C07313=1200.137,5.931,-43.793,-179.713,5.631,148.907
C07314=1200.132,6.181,-43.807,-179.710,5.632,148.906
C07315=1200.127,6.431,-43.821,-179.708,5.632,148.906
C07316=1200.122,6.680,-43.836,-179.705,5.633,148.905
C07317=1200.117,6.929,-43.850,-179.703,5.633,148.904
C07318=1200.112,7.178,-43.865,-179.701,5.633,148.904
C07319=1200.107,7.428,-43.879,-179.698,5.634,148.903
C07320=1200.102,7.678,-43.893,-179.695,5.634,148.902
C07321=1200.097,7.928,-43.907,-179.693,5.635,148.902
C07322=1200.091,8.177,-43.921,-179.691,5.635,148.901
C07323=1200.086,8.426,-43.936,-179.688,5.636,148.900
C07324=1200.081,8.676,-43.950,-179.685,5.636,148.900
C07325=1200.076,8.926,-43.964,-179.683,5.637,148.899
C07326=1200.071,9.175,-43.978,-179.680,5.637,148.898
C07327=1200.066,9.425,-43.993,-179.678,5.638,148.898
C07328=1200.061,9.674,-44.007,-179.675,5.639,148.897
C07329=1200.056,9.923,-44.022,-179.673,5.639,148.897
C07330=1200.051,10.173,-44.036,-179.670,5.639,148.896
C07331=1200.046,10.423,-44.050,-179.668,5.640,148.895
C07332=1200.041,10.673,-44.065,-179.666,5.640,148.895
C07333=1200.036,10.922,-44.079,-179.663,5.641,148.894
C07334=1200.031,11.172,-44.094,-179.660,5.641,148.893
C07335=1200.026,11.421,-44.108,-179.658,5.642,148.893
C07336=1200.021,11.670,-44.123,-179.655,5.642,148.892
C07337=1200.016,11.920,-44.137,-179.652,5.643,148.891
C07338=1200.011,12.170,-44.151,-179.650,5.644,148.891
C07339=1200.006,12.419,-44.166,-179.648,5.644,148.890
C07340=1200.001,12.668,-44.180,-179.645,5.645,148.890
C07341=1199.995,12.918,-44.195,-179.642,5.645,148.889
C07342=1199.990,13.168,-44.210,-179.640,5.646,148.888
C07343=1199.986,13.417,-44.225,-179.637,5.647,148.888
C07344=1199.980,13.666,-44.238,-179.635,5.646,148.887
C07345=1199.975,13.916,-44.253,-179.633,5.647,148.886
C07346=1199.970,14.166,-44.267,-179.630,5.647,148.886
C07347=1199.966,14.415,-44.282,-179.627,5.648,148.885
C07348=1199.960,14.665,-44.297,-179.625,5.649,148.885
C07349=1199.955,14.915,-44.311,-179.623,5.649,148.884
C07350=1199.950,15.164,-44.326,-179.620,5.650,148.883
C07351=1199.945,15.413,-44.340,-179.617,5.650,148.882
C07352=1199.940,15.663,-44.355,-179.615,5.651,148.882
C07353=1199.935,15.912,-44.370,-179.613,5.652,148.881
C07354=1199.930,16.162,-44.385,-179.610,5.652,148.881
C07355=1199.925,16.412,-44.399,-179.607,5.653,148.880
C07356=1199.920,16.661,-44.414,-179.605,5.653,148.879
C07357=1199.916,16.911,-44.428,-179.602,5.654,148.879
C07358=1199.910,17.161,-44.443,-179.600,5.655,148.878
C07359=1199.905,17.410,-44.458,-179.597,5.655,148.877
C07360=1199.900,17.659,-44.472,-179.594,5.656,148.877
C07361=1199.895,17.908,-44.487,-179.592,5.656,148.876
C07362=1199.889,18.158,-44.502,-179.589,5.657,148.875
C07363=1199.884,18.408,-44.516,-179.587,5.657,148.875
C07364=1199.880,18.657,-44.531,-179.584,5.658,148.874
C07365=1199.875,18.906,-44.545,-179.582,5.658,148.874
C07366=1199.869,19.156,-44.561,-179.580,5.658,148.873
C07367=1199.864,19.406,-44.575,-179.577,5.659,148.872
C07368=1199.860,19.655,-44.590,-179.575,5.660,148.872
C07369=1199.854,19.905,-44.605,-179.572,5.660,148.871
C07370=1199.849,20.154,-44.620,-179.570,5.661,148.870
C07371=1199.844,20.403,-44.634,-179.567,5.661,148.870
C07372=1199.839,20.653,-44.650,-179.564,5.662,148.869
C07373=1199.834,20.903,-44.664,-179.562,5.662,148.869
C07374=1199.829,21.152,-44.679,-179.559,5.663,148.868
C07375=1199.824,21.402,-44.694,-179.557,5.663,148.867
C07376=1199.819,21.651,-44.709,-179.554,5.664,148.867
C07377=1199.814,21.900,-44.723,-179.552,5.665,148.866
C07378=1199.809,22.151,-44.739,-179.549,5.665,148.865
C07379=1199.804,22.400,-44.754,-179.547,5.666,148.865
C07380=1199.800,22.649,-44.768,-179.544,5.666,148.864
C07381=1199.794,22.899,-44.783,-179.541,5.667,148.863
C07382=1199.789,23.149,-44.798,-179.539,5.668,148.863
C07383=1199.785,23.398,-44.813,-179.537,5.668,148.862
C07384=1199.779,23.648,-44.828,-179.534,5.669,148.862
C07385=1199.774,23.897,-44.843,-179.531,5.669,148.861
C07386=1199.769,24.147,-44.858,-179.529,5.670,148.860
C07387=1199.764,24.396,-44.873,-179.527,5.671,148.860
C07388=1199.759,24.645,-44.888,-179.524,5.671,148.859
C07389=1199.754,24.895,-44.903,-179.521,5.672,148.858
C07390=1199.749,25.144,-44.918,-179.519,5.672,148.858
C07391=1199.744,25.393,-44.934,-179.516,5.673,148.857
C07392=1199.739,25.643,-44.948,-179.514,5.674,148.857
C07393=1199.735,25.893,-44.963,-179.511,5.674,148.856
C07394=1199.729,26.142,-44.979,-179.508,5.675,148.855
C07395=1199.724,26.392,-44.993,-179.506,5.675,148.855
C07396=1199.719,26.641,-45.009,-179.504,5.676,148.854
C07397=1199.714,26.891,-45.024,-179.501,5.677,148.853
C07398=1199.709,27.141,-45.038,-179.498,5.677,148.853
C07399=1199.704,27.390,-45.053,-179.496,5.678,148.852
C07400=1199.699,27.639,-45.069,-179.494,5.678,148.852
C07401=1199.694,27.888,-45.084,-179.491,5.679,148.851
C07402=1199.689,28.139,-45.099,-179.488,5.680,148.850
C07403=1199.684,28.388,-45.114,-179.486,5.680,148.850
C07404=1199.679,28.656,-45.131,-179.483,5.681,148.849
C07405=1199.674,28.925,-45.147,-179.480,5.681,148.848
C07406=1199.668,29.194,-45.163,-179.478,5.682,148.848
C07407=1199.663,29.462,-45.180,-179.474,5.683,148.847
C07408=1199.657,29.712,-45.195,-179.472,5.684,148.846
C07409=1199.653,29.962,-45.210,-179.470,5.684,148.846
C07410=1199.647,30.211,-45.225,-179.467,5.685,148.845
C07411=1199.642,30.460,-45.241,-179.464,5.685,148.844
C07412=1199.638,30.710,-45.256,-179.462,5.686,148.844
C07413=1199.632,30.960,-45.272,-179.460,5.687,148.843
C07414=1199.628,31.209,-45.287,-179.457,5.687,148.843
C07415=1199.622,31.459,-45.302,-179.454,5.688,148.842
C07416=1199.617,31.708,-45.317,-179.452,5.688,148.841
C07417=1199.613,31.958,-45.333,-179.450,5.689,148.841
C07418=1199.607,32.207,-45.348,-179.447,5.690,148.840
C07419=1199.603,32.456,-45.363,-179.444,5.690,148.839
C07420=1199.597,32.706,-45.379,-179.442,5.691,148.839
C07421=1199.592,32.955,-45.394,-179.439,5.692,148.838
C07422=1199.588,33.205,-45.410,-179.437,5.692,148.838
C07423=1199.582,33.454,-45.425,-179.434,5.693,148.837
C07424=1199.578,33.703,-45.440,-179.431,5.693,148.836
C07425=1199.572,33.954,-45.455,-179.429,5.694,148.836
C07426=1199.567,34.203,-45.470,-179.427,5.695,148.835
C07427=1199.563,34.453,-45.486,-179.424,5.695,148.834
C07428=1199.557,34.702,-45.502,-179.421,5.696,148.834
C07429=1199.552,34.951,-45.517,-179.419,5.697,148.833
C07430=1199.547,35.201,-45.532,-179.417,5.697,148.833
C07431=1199.542,35.451,-45.548,-179.414,5.698,148.832
C07432=1199.538,35.700,-45.563,-179.411,5.698,148.831
C07433=1199.532,35.949,-45.579,-179.408,5.699,148.831
C07434=1199.527,36.199,-45.594,-179.406,5.700,148.830
C07435=1199.523,36.448,-45.610,-179.403,5.701,148.830
C07436=1199.517,36.698,-45.625,-179.401,5.701,148.829
C07437=1199.512,36.947,-45.641,-179.398,5.702,148.828
C07438=1199.507,37.196,-45.656,-179.396,5.703,148.828
C07439=1199.503,37.446,-45.673,-179.393,5.703,148.827
C07440=1199.498,37.695,-45.688,-179.391,5.704,148.826
C07441=1199.492,37.945,-45.704,-179.388,5.704,148.826
C07442=1199.488,38.194,-45.719,-179.386,5.705,148.825
C07443=1199.483,38.444,-45.735,-179.383,5.706,148.825
C07444=1199.477,38.693,-45.750,-179.381,5.706,148.824
C07445=1199.472,38.943,-45.766,-179.378,5.707,148.823
C07446=1199.468,39.192,-45.781,-179.376,5.708,148.823
C07447=1199.463,39.442,-45.797,-179.373,5.708,148.822
C07448=1199.457,39.691,-45.812,-179.370,5.709,148.821
C07449=1199.453,39.941,-45.829,-179.368,5.710,148.821
C07450=1199.448,40.190,-45.844,-179.365,5.711,148.820
C07451=1199.443,40.439,-45.860,-179.362,5.711,148.820
C07452=1199.438,40.689,-45.876,-179.360,5.712,148.819
C07453=1199.432,40.939,-45.891,-179.358,5.713,148.819
C07454=1199.427,41.187,-45.907,-179.355,5.713,148.818
C07455=1199.423,41.437,-45.923,-179.352,5.714,148.817
C07456=1199.418,41.687,-45.938,-179.350,5.714,148.817
C07457=1199.413,41.936,-45.954,-179.348,5.715,148.816
C07458=1199.408,42.186,-45.970,-179.345,5.716,148.815
C07459=1199.403,42.435,-45.986,-179.342,5.716,148.815
C07460=1199.397,42.684,-46.002,-179.340,5.717,148.814
C07461=1199.393,42.934,-46.017,-179.337,5.718,148.814
C07462=1199.388,43.184,-46.033,-179.335,5.718,148.813
C07463=1199.383,43.432,-46.049,-179.332,5.720,148.812
C07464=1199.378,43.682,-46.065,-179.329,5.720,148.812
C07465=1199.373,43.932,-46.081,-179.327,5.721,148.811
C07466=1199.367,44.181,-46.096,-179.324,5.722,148.810
C07467=1199.363,44.431,-46.113,-179.322,5.722,148.810
C07468=1199.358,44.680,-46.128,-179.319,5.723,148.809
C07469=1199.353,44.930,-46.144,-179.317,5.724,148.809
C07470=1199.348,45.179,-46.160,-179.314,5.724,148.808
C07471=1199.343,45.428,-46.176,-179.311,5.725,148.807
C07472=1199.338,45.678,-46.192,-179.309,5.726,148.807
C07473=1199.333,45.927,-46.208,-179.306,5.727,148.806
C07474=1199.328,46.177,-46.224,-179.303,5.727,148.806
C07475=1199.323,46.426,-46.240,-179.301,5.728,148.805
C07476=1199.318,46.675,-46.256,-179.299,5.729,148.804
C07477=1199.313,46.925,-46.272,-179.296,5.729,148.804
C07478=1199.308,47.174,-46.288,-179.293,5.730,148.803
C07479=1199.303,47.424,-46.304,-179.291,5.731,148.803
C07480=1199.298,47.673,-46.320,-179.289,5.731,148.802
C07481=1199.293,47.923,-46.336,-179.286,5.732,148.801
C07482=1199.288,48.173,-46.352,-179.283,5.732,148.801
C07483=1199.284,48.422,-46.368,-179.281,5.734,148.800
C07484=1199.279,48.671,-46.384,-179.278,5.735,148.800
C07485=1199.274,48.920,-46.400,-179.275,5.735,148.799
C07486=1199.269,49.170,-46.416,-179.273,5.736,148.798
C07487=1199.264,49.419,-46.432,-179.271,5.737,148.798
C07488=1199.259,49.669,-46.448,-179.268,5.737,148.797
C07489=1199.254,49.918,-46.464,-179.265,5.738,148.796
C07490=1199.249,50.168,-46.480,-179.263,5.739,148.796
C07491=1199.244,50.417,-46.497,-179.260,5.740,148.795
C07492=1199.239,50.667,-46.513,-179.257,5.740,148.795
C07493=1199.233,50.916,-46.529,-179.255,5.741,148.794
C07494=1199.229,51.166,-46.545,-179.252,5.742,148.794
C07495=1199.224,51.415,-46.562,-179.250,5.742,148.793
C07496=1199.219,51.665,-46.578,-179.248,5.743,148.792
C07497=1199.214,51.914,-46.594,-179.245,5.744,148.792
C07498=1199.209,52.163,-46.611,-179.242,5.744,148.791
C07499=1199.204,52.412,-46.626,-179.239,5.746,148.790
C07500=1199.199,52.662,-46.643,-179.237,5.747,148.790
C07501=1199.194,52.911,-46.659,-179.234,5.747,148.789
C07502=1199.189,53.161,-46.675,-179.232,5.748,148.789
C07503=1199.184,53.410,-46.691,-179.230,5.749,148.788
C07504=1199.180,53.660,-46.707,-179.227,5.749,148.788
C07505=1199.174,53.908,-46.724,-179.224,5.750,148.787
C07506=1199.169,54.159,-46.740,-179.222,5.751,148.786
C07507=1199.164,54.408,-46.757,-179.219,5.752,148.786
C07508=1199.159,54.676,-46.775,-179.216,5.752,148.785
C07509=1199.154,54.945,-46.792,-179.214,5.753,148.784
C07510=1199.149,55.213,-46.810,-179.211,5.754,148.784
C07511=1199.143,55.482,-46.827,-179.208,5.755,148.783
C07512=1199.138,55.732,-46.844,-179.206,5.756,148.783
C07513=1199.133,55.981,-46.860,-179.203,5.756,148.782
C07514=1199.128,56.230,-46.876,-179.200,5.757,148.781
C07515=1199.123,56.479,-46.893,-179.197,5.758,148.781
C07516=1199.119,56.729,-46.909,-179.195,5.759,148.780
C07517=1199.113,56.978,-46.925,-179.192,5.760,148.780
C07518=1199.108,57.228,-46.942,-179.190,5.760,148.779
C07519=1199.104,57.477,-46.959,-179.188,5.761,148.779
C07520=1199.099,57.726,-46.975,-179.185,5.762,148.778
C07521=1199.094,57.976,-46.991,-179.182,5.763,148.777
C07522=1199.088,58.225,-47.008,-179.180,5.764,148.777
C07523=1199.084,58.475,-47.025,-179.177,5.764,148.776
C07524=1199.079,58.724,-47.041,-179.174,5.765,148.775
C07525=1199.074,58.973,-47.058,-179.172,5.766,148.775
C07526=1199.069,59.223,-47.074,-179.170,5.766,148.774
C07527=1199.063,59.472,-47.090,-179.166,5.768,148.774
C07528=1199.059,59.722,-47.107,-179.164,5.769,148.773
C07529=1199.054,59.971,-47.124,-179.162,5.769,148.773
C07530=1199.049,60.220,-47.141,-179.159,5.770,148.772
C07531=1199.044,60.470,-47.157,-179.157,5.771,148.771
C07532=1199.040,60.719,-47.174,-179.154,5.772,148.771
C07533=1199.034,60.969,-47.190,-179.151,5.773,148.770
C07534=1199.029,61.219,-47.207,-179.149,5.773,148.770
C07535=1199.025,61.468,-47.224,-179.146,5.774,148.769
C07536=1199.020,61.717,-47.240,-179.144,5.775,148.768
C07537=1199.014,61.967,-47.257,-179.141,5.775,148.768
C07538=1199.010,62.216,-47.274,-179.138,5.777,148.767
C07539=1199.005,62.465,-47.290,-179.136,5.777,148.767
C07540=1199.000,62.715,-47.307,-179.134,5.778,148.766
C07541=1198.995,62.964,-47.324,-179.131,5.779,148.765
C07542=1198.990,63.213,-47.340,-179.128,5.779,148.765
C07543=1198.985,63.463,-47.358,-179.126,5.781,148.764
C07544=1198.980,63.712,-47.374,-179.123,5.782,148.764
C07545=1198.975,63.961,-47.391,-179.120,5.782,148.763
C07546=1198.970,64.211,-47.408,-179.118,5.783,148.763
C07547=1198.965,64.460,-47.425,-179.115,5.784,148.762
C07548=1198.961,64.710,-47.441,-179.112,5.785,148.761
C07549=1198.955,64.959,-47.458,-179.110,5.786,148.761
C07550=1198.951,65.208,-47.475,-179.107,5.786,148.760
C07551=1198.945,65.458,-47.492,-179.105,5.787,148.760
C07552=1198.940,65.707,-47.508,-179.103,5.788,148.759
C07553=1198.936,65.956,-47.525,-179.100,5.789,148.758
C07554=1198.931,66.206,-47.542,-179.097,5.790,148.758
C07555=1198.926,66.456,-47.559,-179.095,5.791,148.757
C07556=1198.920,66.705,-47.576,-179.092,5.791,148.757
C07557=1198.916,66.954,-47.593,-179.089,5.792,148.756
C07558=1198.912,67.203,-47.610,-179.087,5.794,148.756
C07559=1198.907,67.453,-47.627,-179.084,5.794,148.755
C07560=1198.901,67.702,-47.643,-179.081,5.795,148.754
C07561=1198.896,67.951,-47.661,-179.079,5.796,148.754
C07562=1198.892,68.201,-47.677,-179.076,5.797,148.753
C07563=1198.887,68.451,-47.695,-179.074,5.797,148.753
C07564=1198.882,68.700,-47.711,-179.071,5.798,148.752
C07565=1198.877,68.949,-47.729,-179.069,5.799,148.751
C07566=1198.872,69.198,-47.746,-179.067,5.800,148.751
C07567=1198.867,69.448,-47.763,-179.063,5.801,148.750
C07568=1198.862,69.697,-47.780,-179.061,5.802,148.750
C07569=1198.857,69.947,-47.796,-179.059,5.803,148.749
C07570=1198.852,70.195,-47.814,-179.056,5.803,148.749
C07571=1198.847,70.445,-47.831,-179.053,5.805,148.748
C07572=1198.843,70.695,-47.848,-179.051,5.805,148.748
C07573=1198.837,70.945,-47.865,-179.048,5.806,148.747
C07574=1198.833,71.193,-47.882,-179.045,5.807,148.746
C07575=1198.827,71.442,-47.899,-179.043,5.808,148.746
C07576=1198.823,71.692,-47.916,-179.040,5.809,148.745
C07577=1198.818,71.942,-47.933,-179.038,5.810,148.745
C07578=1198.813,72.191,-47.951,-179.035,5.810,148.744
C07579=1198.808,72.440,-47.968,-179.032,5.812,148.743
C07580=1198.803,72.689,-47.985,-179.030,5.813,148.743
C07581=1198.798,72.938,-48.002,-179.027,5.813,148.742
C07582=1198.793,73.188,-48.019,-179.025,5.814,148.742
C07583=1198.789,73.438,-48.036,-179.022,5.815,148.741
C07584=1198.784,73.687,-48.054,-179.019,5.816,148.741
C07585=1198.779,73.937,-48.071,-179.017,5.817,148.740
C07586=1198.774,74.186,-48.088,-179.015,5.817,148.739
C07587=1198.769,74.435,-48.106,-179.011,5.819,148.739
C07588=1198.763,74.684,-48.123,-179.009,5.820,148.738
C07589=1198.759,74.934,-48.140,-179.007,5.820,148.738
C07590=1198.754,75.183,-48.158,-179.004,5.821,148.737
C07591=1198.749,75.433,-48.174,-179.001,5.823,148.737
C07592=1198.745,75.682,-48.192,-178.999,5.823,148.736
C07593=1198.739,75.931,-48.209,-178.996,5.824,148.736
C07594=1198.735,76.180,-48.227,-178.994,5.825,148.735
C07595=1198.730,76.430,-48.244,-178.991,5.826,148.734
C07596=1198.725,76.680,-48.261,-178.988,5.827,148.734
C07597=1198.719,76.928,-48.279,-178.986,5.827,148.733
C07598=1198.715,77.178,-48.296,-178.983,5.829,148.733
C07599=1198.710,77.427,-48.314,-178.981,5.830,148.732
C07600=1198.705,77.677,-48.331,-178.978,5.830,148.731
C07601=1198.700,77.926,-48.348,-178.976,5.831,148.731
C07602=1198.695,78.176,-48.366,-178.973,5.833,148.730
C07603=1198.690,78.425,-48.384,-178.970,5.833,148.730
C07604=1198.686,78.674,-48.400,-178.968,5.834,148.729
C07605=1198.681,78.923,-48.418,-178.965,5.835,148.729
C07606=1198.676,79.173,-48.436,-178.962,5.836,148.728
C07607=1198.671,79.422,-48.453,-178.960,5.837,148.728
C07608=1198.667,79.671,-48.471,-178.958,5.838,148.727
C07609=1198.661,79.921,-48.488,-178.954,5.839,148.726
C07610=1198.656,80.170,-48.506,-178.952,5.840,148.726
C07611=1198.651,80.420,-48.523,-178.950,5.841,148.725
C07612=1198.646,80.688,-48.542,-178.947,5.842,148.725
C07613=1198.640,80.956,-48.561,-178.944,5.843,148.724
C07614=1198.636,81.224,-48.580,-178.941,5.844,148.723
C07615=1198.630,81.493,-48.599,-178.939,5.845,148.723
C07616=1198.626,81.742,-48.617,-178.936,5.845,148.722
C07617=1198.621,81.992,-48.635,-178.933,5.847,148.722
C07618=1198.615,82.241,-48.652,-178.931,5.848,148.721
C07619=1198.610,82.491,-48.670,-178.928,5.848,148.721
C07620=1198.606,82.739,-48.687,-178.925,5.850,148.720
C07621=1198.601,82.989,-48.704,-178.923,5.851,148.720
C07622=1198.596,83.238,-48.722,-178.920,5.851,148.719
C07623=1198.591,83.488,-48.740,-178.917,5.853,148.718
C07624=1198.586,83.737,-48.758,-178.915,5.853,148.718
C07625=1198.581,83.987,-48.776,-178.913,5.854,148.717
C07626=1198.576,84.236,-48.794,-178.909,5.856,148.717
C07627=1198.571,84.485,-48.812,-178.907,5.857,148.716
C07628=1198.567,84.734,-48.828,-178.905,5.857,148.716
C07629=1198.562,84.984,-48.846,-178.902,5.858,148.715
C07630=1198.557,85.233,-48.864,-178.899,5.860,148.715
C07631=1198.552,85.482,-48.882,-178.897,5.860,148.714
C07632=1198.547,85.731,-48.900,-178.894,5.861,148.713
C07633=1198.542,85.981,-48.917,-178.891,5.862,148.713
C07634=1198.537,86.230,-48.935,-178.889,5.863,148.712
C07635=1198.532,86.479,-48.953,-178.887,5.864,148.712
C07636=1198.527,86.728,-48.971,-178.884,5.866,148.711
C07637=1198.523,86.978,-48.990,-178.881,5.866,148.711
C07638=1198.518,87.227,-49.008,-178.879,5.867,148.710
C07639=1198.513,87.477,-49.025,-178.876,5.868,148.710
C07640=1198.508,87.726,-49.043,-178.873,5.869,148.709
C07641=1198.504,87.975,-49.060,-178.871,5.870,148.709
C07642=1198.499,88.224,-49.078,-178.868,5.871,148.708
C07643=1198.494,88.474,-49.096,-178.866,5.872,148.707
C07644=1198.489,88.723,-49.114,-178.863,5.873,148.707
C07645=1198.484,88.972,-49.132,-178.860,5.875,148.706
C07646=1198.479,89.221,-49.150,-178.858,5.875,148.706
C07647=1198.475,89.471,-49.169,-178.855,5.876,148.705
C07648=1198.470,89.720,-49.187,-178.852,5.877,148.705
C07649=1198.464,89.970,-49.204,-178.850,5.878,148.704
C07650=1198.459,90.219,-49.222,-178.847,5.880,148.704
C07651=1198.454,90.469,-49.240,-178.845,5.880,148.703
C07652=1198.449,90.718,-49.258,-178.842,5.881,148.703
C07653=1198.444,90.967,-49.276,-178.839,5.883,148.702
C07654=1198.439,91.216,-49.294,-178.837,5.884,148.702
C07655=1198.435,91.466,-49.313,-178.834,5.884,148.701
C07656=1198.430,91.715,-49.331,-178.832,5.886,148.700
C07657=1198.425,91.964,-49.349,-178.829,5.886,148.700
C07658=1198.420,92.214,-49.367,-178.826,5.887,148.699
C07659=1198.415,92.463,-49.385,-178.824,5.889,148.699
C07660=1198.411,92.711,-49.403,-178.821,5.889,148.698
C07661=1198.407,92.961,-49.422,-178.818,5.891,148.698
C07662=1198.402,93.210,-49.440,-178.816,5.892,148.697
C07663=1198.397,93.460,-49.458,-178.814,5.893,148.697
C07664=1198.391,93.709,-49.476,-178.810,5.894,148.696
C07665=1198.386,93.958,-49.494,-178.808,5.895,148.696
C07666=1198.382,94.208,-49.512,-178.806,5.895,148.695
C07667=1198.377,94.457,-49.530,-178.803,5.897,148.694
C07668=1198.372,94.706,-49.548,-178.800,5.898,148.694
C07669=1198.367,94.956,-49.566,-178.798,5.899,148.693
C07670=1198.362,95.204,-49.585,-178.795,5.900,148.693
C07671=1198.357,95.454,-49.604,-178.793,5.901,148.692
C07672=1198.353,95.704,-49.622,-178.790,5.902,148.692
C07673=1198.348,95.953,-49.640,-178.787,5.903,148.691
C07674=1198.343,96.202,-49.658,-178.785,5.904,148.691
C07675=1198.338,96.452,-49.676,-178.782,5.905,148.690
C07676=1198.333,96.701,-49.696,-178.780,5.906,148.690
C07677=1198.328,96.950,-49.714,-178.776,5.908,148.689
C07678=1198.323,97.199,-49.732,-178.774,5.908,148.689
C07679=1198.319,97.449,-49.750,-178.772,5.909,148.688
C07680=1198.314,97.697,-49.769,-178.769,5.911,148.687
C07681=1198.309,97.947,-49.787,-178.766,5.911,148.687
C07682=1198.304,98.196,-49.805,-178.764,5.913,148.686
C07683=1198.299,98.446,-49.824,-178.761,5.914,148.686
C07684=1198.295,98.694,-49.842,-178.759,5.915,148.685
C07685=1198.289,98.944,-49.861,-178.756,5.916,148.685
C07686=1198.284,99.193,-49.879,-178.754,5.917,148.684
C07687=1198.280,99.442,-49.898,-178.750,5.918,148.684
C07688=1198.275,99.692,-49.916,-178.748,5.919,148.683
C07689=1198.270,99.941,-49.934,-178.746,5.920,148.683
C07690=1198.265,100.191,-49.953,-178.743,5.922,148.682
C07691=1198.261,100.440,-49.971,-178.740,5.922,148.682
C07692=1198.255,100.689,-49.990,-178.738,5.924,148.681
C07693=1198.251,100.938,-50.009,-178.735,5.924,148.680
C07694=1198.246,101.187,-50.027,-178.733,5.925,148.680
C07695=1198.241,101.437,-50.046,-178.730,5.927,148.679
C07696=1198.237,101.686,-50.065,-178.728,5.928,148.679
C07697=1198.232,101.935,-50.083,-178.724,5.929,148.678
C07698=1198.226,102.184,-50.102,-178.722,5.930,148.678
C07699=1198.222,102.434,-50.120,-178.719,5.931,148.677
C07700=1198.217,102.683,-50.138,-178.717,5.932,148.677
C07701=1198.212,102.932,-50.158,-178.714,5.933,148.676
C07702=1198.207,103.182,-50.176,-178.712,5.935,148.676
C07703=1198.203,103.431,-50.195,-178.709,5.935,148.675
C07704=1198.197,103.680,-50.213,-178.706,5.937,148.675
C07705=1198.193,103.929,-50.232,-178.704,5.938,148.674
C07706=1198.188,104.179,-50.251,-178.701,5.939,148.674
C07707=1198.183,104.427,-50.270,-178.699,5.940,148.673
C07708=1198.179,104.677,-50.288,-178.696,5.941,148.673
C07709=1198.173,104.926,-50.307,-178.694,5.943,148.672
C07710=1198.169,105.176,-50.325,-178.691,5.943,148.672
C07711=1198.164,105.425,-50.345,-178.688,5.945,148.671
C07712=1198.159,105.674,-50.363,-178.686,5.946,148.671
C07713=1198.154,105.924,-50.382,-178.683,5.947,148.670
C07714=1198.149,106.173,-50.400,-178.680,5.948,148.670
C07715=1198.144,106.421,-50.419,-178.678,5.950,148.669
C07716=1198.139,106.691,-50.439,-178.675,5.950,148.668
C07717=1198.134,106.959,-50.460,-178.672,5.952,148.668
C07718=1198.129,107.227,-50.480,-178.670,5.953,148.667
C07719=1198.124,107.495,-50.501,-178.666,5.954,148.667
C07720=1198.118,107.744,-50.520,-178.664,5.956,148.666
C07721=1198.114,107.994,-50.538,-178.661,5.956,148.666
C07722=1198.109,108.243,-50.558,-178.658,5.958,148.665
C07723=1198.105,108.492,-50.577,-178.656,5.959,148.665
C07724=1198.099,108.742,-50.595,-178.654,5.960,148.664
C07725=1198.095,108.991,-50.614,-178.651,5.961,148.664
C07726=1198.090,109.240,-50.634,-178.648,5.962,148.663
C07727=1198.085,109.490,-50.652,-178.645,5.963,148.663
C07728=1198.080,109.739,-50.671,-178.643,5.964,148.662
C07729=1198.075,109.987,-50.690,-178.640,5.966,148.662
C07730=1198.070,110.237,-50.709,-178.638,5.967,148.661
C07731=1198.066,110.486,-50.728,-178.635,5.968,148.661
C07732=1198.061,110.736,-50.747,-178.632,5.969,148.660
C07733=1198.056,110.984,-50.767,-178.630,5.971,148.660
C07734=1198.051,111.234,-50.785,-178.627,5.971,148.659
C07735=1198.046,111.483,-50.804,-178.624,5.973,148.659
C07736=1198.042,111.732,-50.823,-178.622,5.974,148.658
C07737=1198.037,111.981,-50.843,-178.619,5.975,148.658
C07738=1198.032,112.231,-50.862,-178.617,5.976,148.657
C07739=1198.027,112.480,-50.880,-178.614,5.978,148.657
C07740=1198.022,112.730,-50.900,-178.612,5.979,148.656
C07741=1198.018,112.978,-50.918,-178.609,5.980,148.656
C07742=1198.013,113.228,-50.938,-178.606,5.981,148.655
C07743=1198.008,113.477,-50.957,-178.603,5.982,148.655
C07744=1198.004,113.726,-50.976,-178.601,5.983,148.654
C07745=1197.999,113.976,-50.995,-178.598,5.985,148.654
C07746=1197.993,114.225,-51.015,-178.596,5.986,148.653
C07747=1197.989,114.474,-51.034,-178.593,5.987,148.653
C07748=1197.984,114.723,-51.053,-178.590,5.988,148.652
C07749=1197.979,114.973,-51.073,-178.588,5.990,148.652
C07750=1197.975,115.221,-51.091,-178.585,5.990,148.651
C07751=1197.970,115.471,-51.111,-178.582,5.992,148.651
C07752=1197.964,115.720,-51.130,-178.580,5.993,148.650
C07753=1197.960,115.969,-51.150,-178.577,5.994,148.650
C07754=1197.955,116.218,-51.169,-178.575,5.995,148.649
C07755=1197.950,116.467,-51.188,-178.572,5.997,148.649
C07756=1197.946,116.717,-51.208,-178.570,5.998,148.648
C07757=1197.941,116.965,-51.227,-178.567,5.999,148.648
C07758=1197.936,117.215,-51.246,-178.564,6.000,148.647
C07759=1197.931,117.464,-51.266,-178.562,6.002,148.647
C07760=1197.926,117.713,-51.285,-178.559,6.002,148.646
C07761=1197.921,117.963,-51.305,-178.556,6.004,148.646
C07762=1197.917,118.212,-51.324,-178.554,6.005,148.645
C07763=1197.912,118.461,-51.343,-178.551,6.006,148.645
C07764=1197.907,118.710,-51.363,-178.549,6.007,148.644
C07765=1197.902,118.960,-51.382,-178.546,6.009,148.644
C07766=1197.898,119.209,-51.401,-178.544,6.010,148.643
C07767=1197.893,119.458,-51.421,-178.541,6.012,148.643
C07768=1197.888,119.707,-51.440,-178.538,6.012,148.642
C07769=1197.883,119.957,-51.460,-178.536,6.014,148.642
C07770=1197.878,120.206,-51.479,-178.533,6.014,148.641
C07771=1197.873,120.455,-51.499,-178.530,6.016,148.641
C07772=1197.869,120.704,-51.519,-178.528,6.017,148.640
C07773=1197.864,120.953,-51.538,-178.525,6.019,148.640
C07774=1197.859,121.202,-51.558,-178.522,6.020,148.639
C07775=1197.855,121.452,-51.577,-178.520,6.021,148.639
C07776=1197.849,121.701,-51.597,-178.517,6.023,148.638
C07777=1197.844,121.950,-51.616,-178.515,6.024,148.638
C07778=1197.840,122.199,-51.637,-178.512,6.025,148.637
C07779=1197.835,122.448,-51.655,-178.510,6.026,148.637
C07780=1197.831,122.697,-51.675,-178.506,6.027,148.636
C07781=1197.826,122.947,-51.695,-178.504,6.028,148.636
C07782=1197.821,123.195,-51.715,-178.502,6.030,148.635
C07783=1197.816,123.445,-51.734,-178.498,6.031,148.635
C07784=1197.811,123.694,-51.754,-178.496,6.032,148.634
C07785=1197.806,123.943,-51.773,-178.494,6.034,148.634
C07786=1197.802,124.192,-51.794,-178.491,6.035,148.633
C07787=1197.797,124.442,-51.813,-178.488,6.037,148.633
C07788=1197.792,124.691,-51.833,-178.486,6.037,148.632
C07789=1197.787,124.940,-51.852,-178.483,6.039,148.632
C07790=1197.782,125.189,-51.873,-178.481,6.040,148.631
C07791=1197.778,125.439,-51.892,-178.478,6.041,148.631
C07792=1197.772,125.688,-51.912,-178.475,6.043,148.630
C07793=1197.768,125.936,-51.932,-178.473,6.044,148.630
C07794=1197.763,126.186,-51.952,-178.470,6.045,148.629
C07795=1197.758,126.436,-51.971,-178.468,6.046,148.629
C07796=1197.753,126.684,-51.991,-178.465,6.048,148.629
C07797=1197.749,126.933,-52.011,-178.462,6.049,148.628
C07798=1197.744,127.182,-52.031,-178.460,6.050,148.628
C07799=1197.739,127.432,-52.051,-178.457,6.052,148.627
C07800=1197.735,127.682,-52.071,-178.454,6.053,148.627
C07801=1197.730,127.930,-52.091,-178.452,6.055,148.626
C07802=1197.725,128.179,-52.110,-178.449,6.055,148.626
C07803=1197.720,128.428,-52.131,-178.446,6.057,148.625
C07804=1197.716,128.678,-52.150,-178.444,6.059,148.625
C07805=1197.711,128.927,-52.171,-178.441,6.059,148.624
C07806=1197.706,129.176,-52.190,-178.438,6.061,148.624
C07807=1197.701,129.425,-52.210,-178.436,6.062,148.623
C07808=1197.697,129.674,-52.230,-178.433,6.063,148.623
C07809=1197.692,129.923,-52.250,-178.430,6.065,148.622
C07810=1197.688,130.173,-52.270,-178.428,6.066,148.622
C07811=1197.682,130.421,-52.290,-178.425,6.068,148.621
C07812=1197.678,130.671,-52.310,-178.423,6.069,148.621
C07813=1197.673,130.920,-52.331,-178.420,6.070,148.621
C07814=1197.668,131.169,-52.350,-178.417,6.072,148.620
C07815=1197.663,131.418,-52.371,-178.415,6.073,148.620
C07816=1197.659,131.668,-52.390,-178.412,6.074,148.619
C07817=1197.654,131.916,-52.410,-178.410,6.075,148.618
C07818=1197.649,132.165,-52.431,-178.407,6.077,148.618
C07819=1197.644,132.415,-52.450,-178.404,6.079,148.618
C07820=1197.639,132.683,-52.473,-178.402,6.079,148.617
C07821=1197.633,132.952,-52.494,-178.399,6.081,148.617
C07822=1197.629,133.221,-52.515,-178.396,6.082,148.616
C07823=1197.623,133.489,-52.538,-178.393,6.084,148.616
C07824=1197.619,133.738,-52.558,-178.391,6.085,148.615
C07825=1197.614,133.987,-52.578,-178.388,6.087,148.615
C07826=1197.610,134.236,-52.598,-178.385,6.088,148.614
C07827=1197.605,134.485,-52.619,-178.383,6.089,148.614
C07828=1197.600,134.735,-52.639,-178.380,6.091,148.613
C07829=1197.595,134.984,-52.659,-178.377,6.092,148.613
C07830=1197.591,135.233,-52.680,-178.375,6.093,148.612
C07831=1197.586,135.483,-52.699,-178.372,6.095,148.612
C07832=1197.580,135.731,-52.720,-178.370,6.096,148.611
C07833=1197.576,135.980,-52.740,-178.367,6.098,148.611
C07834=1197.571,136.229,-52.761,-178.364,6.099,148.610
C07835=1197.567,136.479,-52.780,-178.362,6.100,148.610
C07836=1197.561,136.728,-52.801,-178.359,6.102,148.610
C07837=1197.557,136.977,-52.822,-178.356,6.103,148.609
C07838=1197.553,137.226,-52.842,-178.354,6.104,148.609
C07839=1197.547,137.475,-52.863,-178.351,6.106,148.608
C07840=1197.543,137.725,-52.883,-178.348,6.108,148.608
C07841=1197.538,137.974,-52.903,-178.346,6.108,148.607
C07842=1197.533,138.223,-52.924,-178.343,6.110,148.607
C07843=1197.529,138.472,-52.944,-178.341,6.112,148.606
C07844=1197.524,138.721,-52.965,-178.338,6.112,148.606
C07845=1197.519,138.970,-52.986,-178.335,6.114,148.605
C07846=1197.515,139.219,-53.006,-178.333,6.116,148.605
C07847=1197.510,139.469,-53.026,-178.330,6.117,148.605
C07848=1197.505,139.718,-53.047,-178.327,6.118,148.604
C07849=1197.500,139.967,-53.067,-178.325,6.120,148.604
C07850=1197.496,140.216,-53.087,-178.322,6.121,148.603
C07851=1197.491,140.465,-53.108,-178.320,6.123,148.603
C07852=1197.486,140.714,-53.129,-178.317,6.124,148.602
C07853=1197.481,140.963,-53.150,-178.314,6.125,148.602
C07854=1197.477,141.212,-53.170,-178.312,6.127,148.602
C07855=1197.472,141.461,-53.190,-178.309,6.128,148.601
C07856=1197.467,141.710,-53.211,-178.307,6.129,148.601
C07857=1197.462,141.959,-53.232,-178.304,6.131,148.600
C07858=1197.457,142.209,-53.253,-178.301,6.133,148.600
C07859=1197.453,142.458,-53.273,-178.299,6.133,148.599
C07860=1197.448,142.706,-53.294,-178.296,6.135,148.599
C07861=1197.443,142.956,-53.314,-178.293,6.137,148.598
C07862=1197.439,143.205,-53.335,-178.291,6.138,148.598
C07863=1197.434,143.454,-53.356,-178.288,6.139,148.597
C07864=1197.429,143.703,-53.376,-178.285,6.141,148.597
C07865=1197.424,143.952,-53.397,-178.283,6.142,148.597
C07866=1197.420,144.201,-53.418,-178.280,6.144,148.596
C07867=1197.414,144.450,-53.438,-178.277,6.145,148.596
C07868=1197.410,144.699,-53.459,-178.275,6.146,148.595
C07869=1197.405,144.948,-53.481,-178.272,6.148,148.595
C07870=1197.401,145.198,-53.501,-178.270,6.150,148.594
C07871=1197.396,145.447,-53.522,-178.267,6.150,148.594
C07872=1197.392,145.696,-53.543,-178.265,6.152,148.593
C07873=1197.386,145.945,-53.564,-178.262,6.154,148.593
C07874=1197.382,146.194,-53.584,-178.259,6.156,148.593
C07875=1197.377,146.443,-53.606,-178.257,6.156,148.592
C07876=1197.373,146.692,-53.626,-178.254,6.158,148.592
C07877=1197.368,146.941,-53.647,-178.251,6.160,148.591
C07878=1197.362,147.190,-53.668,-178.249,6.161,148.591
C07879=1197.358,147.439,-53.688,-178.246,6.162,148.590
C07880=1197.354,147.688,-53.710,-178.243,6.164,148.590
C07881=1197.349,147.937,-53.731,-178.241,6.166,148.590
C07882=1197.344,148.187,-53.752,-178.238,6.167,148.589
C07883=1197.339,148.436,-53.773,-178.236,6.169,148.589
C07884=1197.335,148.684,-53.794,-178.233,6.170,148.588
C07885=1197.330,148.933,-53.815,-178.230,6.171,148.588
C07886=1197.325,149.182,-53.835,-178.228,6.173,148.587
C07887=1197.321,149.432,-53.856,-178.225,6.175,148.587
C07888=1197.316,149.681,-53.878,-178.222,6.176,148.586
C07889=1197.311,149.930,-53.898,-178.220,6.177,148.586
C07890=1197.306,150.179,-53.919,-178.217,6.179,148.586
C07891=1197.301,150.428,-53.941,-178.214,6.181,148.585
C07892=1197.297,150.677,-53.962,-178.212,6.182,148.585
C07893=1197.292,150.927,-53.983,-178.209,6.183,148.584
C07894=1197.287,151.175,-54.005,-178.207,6.185,148.584
C07895=1197.283,151.424,-54.025,-178.204,6.187,148.583
C07896=1197.278,151.673,-54.047,-178.202,6.187,148.583
C07897=1197.273,151.922,-54.068,-178.199,6.189,148.583
C07898=1197.268,152.172,-54.089,-178.196,6.191,148.582
C07899=1197.264,152.421,-54.110,-178.193,6.192,148.582
C07900=1197.259,152.670,-54.131,-178.191,6.193,148.581
C07901=1197.254,152.918,-54.153,-178.188,6.195,148.581
C07902=1197.250,153.167,-54.173,-178.186,6.197,148.581
C07903=1197.245,153.417,-54.195,-178.183,6.198,148.580
C07904=1197.240,153.666,-54.216,-178.180,6.199,148.580
C07905=1197.235,153.915,-54.238,-178.178,6.201,148.579
C07906=1197.230,154.164,-54.259,-178.175,6.203,148.579
C07907=1197.227,154.413,-54.280,-178.172,6.205,148.578
C07908=1197.221,154.662,-54.301,-178.170,6.205,148.578
C07909=1197.217,154.911,-54.323,-178.167,6.207,148.577
C07910=1197.211,155.160,-54.344,-178.164,6.209,148.577
C07911=1197.208,155.409,-54.365,-178.162,6.211,148.577
C07912=1197.203,155.658,-54.386,-178.160,6.212,148.576
C07913=1197.198,155.907,-54.408,-178.157,6.213,148.576
C07914=1197.193,156.156,-54.429,-178.154,6.215,148.575
C07915=1197.188,156.406,-54.451,-178.151,6.217,148.575
C07916=1197.184,156.654,-54.473,-178.149,6.218,148.575
C07917=1197.179,156.903,-54.493,-178.146,6.219,148.574
C07918=1197.175,157.153,-54.515,-178.144,6.221,148.574
C07919=1197.170,157.402,-54.536,-178.141,6.223,148.573
C07920=1197.165,157.650,-54.558,-178.138,6.224,148.573
C07921=1197.161,157.900,-54.580,-178.136,6.225,148.572
C07922=1197.155,158.149,-54.601,-178.133,6.227,148.572
C07923=1197.151,158.398,-54.622,-178.130,6.229,148.572
C07924=1197.146,158.667,-54.645,-178.127,6.230,148.571
C07925=1197.141,158.935,-54.669,-178.125,6.232,148.571
C07926=1197.136,159.205,-54.692,-178.122,6.234,148.570
C07927=1197.130,159.474,-54.715,-178.119,6.235,148.570
C07928=1197.125,159.723,-54.737,-178.116,6.237,148.569
C07929=1197.121,159.972,-54.759,-178.113,6.239,148.569
C07930=1197.116,160.220,-54.781,-178.111,6.240,148.569
C07931=1197.111,160.470,-54.802,-178.109,6.242,148.568
C07932=1197.108,160.719,-54.823,-178.106,6.244,148.568
C07933=1197.103,160.967,-54.845,-178.103,6.245,148.568
C07934=1197.099,161.217,-54.867,-178.100,6.247,148.567
C07935=1197.093,161.466,-54.888,-178.098,6.248,148.567
C07936=1197.088,161.715,-54.909,-178.095,6.250,148.566
C07937=1197.084,161.964,-54.932,-178.093,6.251,148.566
C07938=1197.079,162.213,-54.953,-178.090,6.253,148.565
C07939=1197.074,162.461,-54.975,-178.087,6.255,148.565
C07940=1197.070,162.711,-54.997,-178.085,6.256,148.565
C07941=1197.065,162.960,-55.018,-178.082,6.257,148.564
C07942=1197.061,163.209,-55.040,-178.079,6.259,148.564
C07943=1197.056,163.458,-55.062,-178.077,6.261,148.563
C07944=1197.051,163.707,-55.083,-178.074,6.263,148.563
C07945=1197.046,163.956,-55.106,-178.071,6.265,148.563
C07946=1197.041,164.205,-55.128,-178.069,6.265,148.562
C07947=1197.037,164.454,-55.150,-178.067,6.267,148.562
C07948=1197.032,164.703,-55.171,-178.064,6.269,148.562
C07949=1197.028,164.952,-55.193,-178.061,6.271,148.561
C07950=1197.023,165.201,-55.215,-178.058,6.272,148.561
C07951=1197.019,165.450,-55.237,-178.056,6.273,148.560
C07952=1197.014,165.699,-55.259,-178.053,6.275,148.560
C07953=1197.009,165.947,-55.281,-178.051,6.277,148.559
C07954=1197.005,166.197,-55.303,-178.048,6.279,148.559
C07955=1197.000,166.445,-55.324,-178.045,6.280,148.559
C07956=1196.995,166.695,-55.346,-178.043,6.282,148.558
C07957=1196.990,166.944,-55.369,-178.041,6.283,148.558
C07958=1196.986,167.193,-55.391,-178.037,6.285,148.557
C07959=1196.981,167.442,-55.412,-178.035,6.286,148.557
C07960=1196.976,167.691,-55.434,-178.032,6.288,148.557
C07961=1196.972,167.940,-55.456,-178.029,6.290,148.556
C07962=1196.967,168.189,-55.478,-178.027,6.292,148.556
C07963=1196.962,168.438,-55.500,-178.024,6.294,148.556
C07964=1196.957,168.687,-55.522,-178.022,6.295,148.555
C07965=1196.953,168.935,-55.545,-178.019,6.296,148.555
C07966=1196.949,169.185,-55.567,-178.017,6.298,148.554
C07967=1196.944,169.433,-55.589,-178.014,6.300,148.554
C07968=1196.939,169.683,-55.611,-178.011,6.302,148.554
C07969=1196.934,169.932,-55.633,-178.008,6.303,148.553
C07970=1196.930,170.181,-55.655,-178.005,6.305,148.553
C07971=1196.925,170.430,-55.677,-178.003,6.306,148.552
C07972=1196.920,170.679,-55.700,-178.001,6.308,148.552
C07973=1196.915,170.927,-55.722,-177.998,6.310,148.552
C07974=1196.911,171.177,-55.744,-177.995,6.311,148.551
C07975=1196.907,171.426,-55.766,-177.993,6.313,148.551
C07976=1196.901,171.674,-55.789,-177.990,6.315,148.551
C07977=1196.897,171.924,-55.811,-177.987,6.317,148.550
C07978=1196.892,172.172,-55.832,-177.985,6.319,148.550
C07979=1196.888,172.422,-55.854,-177.982,6.319,148.549
C07980=1196.883,172.670,-55.877,-177.980,6.321,148.549
C07981=1196.878,172.919,-55.900,-177.977,6.323,148.549
C07982=1196.874,173.169,-55.922,-177.974,6.325,148.548
C07983=1196.869,173.417,-55.945,-177.971,6.326,148.548
C07984=1196.864,173.666,-55.967,-177.969,6.328,148.547
C07985=1196.860,173.915,-55.988,-177.966,6.330,148.547
C07986=1196.855,174.164,-56.012,-177.963,6.332,148.547
C07987=1196.851,174.413,-56.034,-177.961,6.333,148.546
C07988=1196.846,174.662,-56.055,-177.959,6.334,148.546
C07989=1196.841,174.911,-56.079,-177.956,6.336,148.546
C07990=1196.836,175.160,-56.100,-177.953,6.338,148.545
C07991=1196.831,175.409,-56.123,-177.951,6.340,148.545
C07992=1196.827,175.658,-56.146,-177.948,6.342,148.544
C07993=1196.822,175.907,-56.168,-177.945,6.343,148.544
C07994=1196.818,176.156,-56.191,-177.943,6.345,148.544
C07995=1196.813,176.405,-56.213,-177.940,6.347,148.543
C07996=1196.808,176.653,-56.236,-177.937,6.349,148.543
C07997=1196.804,176.903,-56.258,-177.935,6.350,148.543
C07998=1196.800,177.151,-56.281,-177.932,6.352,148.542
C07999=1196.794,177.400,-56.303,-177.930,6.353,148.542
C08000=1196.790,177.649,-56.326,-177.927,6.355,148.542
C08001=1196.785,177.899,-56.348,-177.924,6.357,148.541
C08002=1196.781,178.147,-56.371,-177.922,6.359,148.541
C08003=1196.776,178.396,-56.393,-177.919,6.360,148.540
C08004=1196.772,178.645,-56.416,-177.916,6.362,148.540
C08005=1196.766,178.894,-56.439,-177.913,6.364,148.540
C08006=1196.762,179.143,-56.461,-177.911,6.366,148.539
C08007=1196.757,179.392,-56.484,-177.908,6.367,148.539
C08008=1196.753,179.640,-56.506,-177.905,6.369,148.538
C08009=1196.748,179.889,-56.530,-177.903,6.370,148.538
C08010=1196.744,180.139,-56.552,-177.901,6.372,148.538
C08011=1196.739,180.388,-56.575,-177.898,6.374,148.537
C08012=1196.734,180.636,-56.597,-177.895,6.376,148.537
C08013=1196.729,180.885,-56.620,-177.893,6.377,148.537
C08014=1196.725,181.134,-56.643,-177.890,6.379,148.536
C08015=1196.720,181.384,-56.666,-177.887,6.381,148.536
C08016=1196.716,181.632,-56.688,-177.885,6.383,148.536
C08017=1196.711,181.881,-56.711,-177.882,6.385,148.535
C08018=1196.706,182.131,-56.734,-177.879,6.386,148.535
C08019=1196.702,182.379,-56.757,-177.877,6.388,148.535
C08020=1196.697,182.628,-56.780,-177.874,6.390,148.534
C08021=1196.693,182.876,-56.802,-177.871,6.392,148.534
C08022=1196.688,183.126,-56.825,-177.869,6.394,148.533
C08023=1196.684,183.375,-56.848,-177.866,6.395,148.533
C08024=1196.679,183.623,-56.871,-177.863,6.397,148.533
C08025=1196.674,183.872,-56.894,-177.861,6.398,148.532
C08026=1196.670,184.121,-56.916,-177.858,6.400,148.532
C08027=1196.665,184.370,-56.940,-177.856,6.402,148.532
C08028=1196.660,184.640,-56.965,-177.853,6.404,148.531
C08029=1196.655,184.910,-56.989,-177.850,6.406,148.531
C08030=1196.650,185.179,-57.014,-177.847,6.408,148.531
C08031=1196.646,185.448,-57.039,-177.845,6.410,148.530
C08032=1196.641,185.698,-57.062,-177.842,6.412,148.530
C08033=1196.635,185.946,-57.085,-177.839,6.414,148.530
C08034=1196.631,186.195,-57.108,-177.837,6.415,148.529
C08035=1196.627,186.444,-57.131,-177.834,6.417,148.529
C08036=1196.622,186.693,-57.154,-177.831,6.419,148.528
C08037=1196.617,186.942,-57.178,-177.829,6.421,148.528
C08038=1196.613,187.191,-57.201,-177.826,6.423,148.528
C08039=1196.608,187.440,-57.224,-177.823,6.424,148.527
C08040=1196.603,187.688,-57.247,-177.821,6.426,148.527
C08041=1196.598,187.937,-57.270,-177.818,6.428,148.527
C08042=1196.595,188.186,-57.293,-177.815,6.430,148.526
C08043=1196.590,188.435,-57.316,-177.813,6.432,148.526
C08044=1196.585,188.685,-57.339,-177.810,6.433,148.526
C08045=1196.580,188.934,-57.362,-177.807,6.435,148.525
C08046=1196.576,189.182,-57.385,-177.805,6.437,148.525
C08047=1196.571,189.430,-57.409,-177.802,6.439,148.525
C08048=1196.566,189.679,-57.432,-177.799,6.441,148.524
C08049=1196.562,189.928,-57.456,-177.797,6.442,148.524
C08050=1196.557,190.177,-57.479,-177.794,6.444,148.524
C08051=1196.552,190.426,-57.502,-177.791,6.446,148.523
C08052=1196.548,190.675,-57.525,-177.789,6.448,148.523
C08053=1196.544,190.924,-57.548,-177.787,6.450,148.523
C08054=1196.539,191.173,-57.572,-177.784,6.452,148.522
C08055=1196.534,191.422,-57.595,-177.781,6.454,148.522
C08056=1196.530,191.671,-57.618,-177.779,6.455,148.522
C08057=1196.525,191.920,-57.642,-177.776,6.457,148.521
C08058=1196.520,192.168,-57.665,-177.773,6.459,148.521
C08059=1196.516,192.416,-57.688,-177.771,6.461,148.521
C08060=1196.511,192.666,-57.712,-177.768,6.463,148.520
C08061=1196.507,192.915,-57.735,-177.765,6.464,148.520
C08062=1196.502,193.164,-57.758,-177.763,6.466,148.520
C08063=1196.497,193.413,-57.782,-177.760,6.468,148.519
C08064=1196.492,193.662,-57.805,-177.757,6.470,148.519
C08065=1196.488,193.910,-57.829,-177.755,6.472,148.519
C08066=1196.483,194.159,-57.853,-177.752,6.473,148.518
C08067=1196.479,194.408,-57.876,-177.749,6.475,148.518
C08068=1196.474,194.657,-57.899,-177.747,6.477,148.518
C08069=1196.470,194.906,-57.923,-177.744,6.479,148.517
C08070=1196.465,195.155,-57.947,-177.742,6.481,148.517
C08071=1196.460,195.404,-57.970,-177.739,6.483,148.517
C08072=1196.455,195.653,-57.993,-177.736,6.485,148.516
C08073=1196.451,195.901,-58.017,-177.734,6.486,148.516
C08074=1196.446,196.150,-58.041,-177.731,6.488,148.516
C08075=1196.442,196.399,-58.064,-177.729,6.490,148.515
C08076=1196.437,196.648,-58.088,-177.726,6.492,148.515
C08077=1196.433,196.897,-58.112,-177.723,6.494,148.515
C08078=1196.428,197.146,-58.135,-177.721,6.495,148.514
C08079=1196.423,197.394,-58.159,-177.718,6.498,148.514
C08080=1196.419,197.643,-58.182,-177.715,6.500,148.514
C08081=1196.414,197.891,-58.206,-177.712,6.502,148.513
C08082=1196.410,198.141,-58.230,-177.710,6.504,148.513
C08083=1196.405,198.390,-58.253,-177.707,6.506,148.513
C08084=1196.401,198.638,-58.277,-177.705,6.508,148.512
C08085=1196.396,198.888,-58.301,-177.702,6.509,148.512
C08086=1196.392,199.136,-58.325,-177.699,6.511,148.512
C08087=1196.387,199.385,-58.348,-177.697,6.513,148.511
C08088=1196.383,199.634,-58.373,-177.694,6.515,148.511
C08089=1196.378,199.883,-58.396,-177.692,6.517,148.511
C08090=1196.374,200.131,-58.420,-177.689,6.519,148.511
C08091=1196.368,200.380,-58.444,-177.686,6.521,148.510
C08092=1196.364,200.629,-58.468,-177.684,6.522,148.510
C08093=1196.359,200.878,-58.491,-177.681,6.524,148.510
C08094=1196.355,201.126,-58.515,-177.678,6.526,148.509
C08095=1196.350,201.375,-58.539,-177.676,6.528,148.509
C08096=1196.346,201.624,-58.563,-177.673,6.531,148.509
C08097=1196.342,201.873,-58.587,-177.670,6.533,148.508
C08098=1196.337,202.122,-58.611,-177.668,6.534,148.508
C08099=1196.332,202.371,-58.635,-177.665,6.536,148.508
C08100=1196.328,202.620,-58.659,-177.662,6.538,148.507
C08101=1196.323,202.868,-58.683,-177.660,6.540,148.507
C08102=1196.319,203.116,-58.707,-177.657,6.542,148.507
C08103=1196.314,203.366,-58.731,-177.655,6.544,148.507
C08104=1196.310,203.615,-58.755,-177.652,6.546,148.506
C08105=1196.305,203.864,-58.779,-177.650,6.547,148.506
C08106=1196.300,204.112,-58.803,-177.647,6.549,148.506
C08107=1196.296,204.361,-58.827,-177.644,6.551,148.505
C08108=1196.291,204.609,-58.851,-177.641,6.554,148.505
C08109=1196.287,204.859,-58.875,-177.638,6.556,148.505
C08110=1196.282,205.108,-58.899,-177.636,6.558,148.504
C08111=1196.277,205.356,-58.924,-177.634,6.559,148.504
C08112=1196.273,205.605,-58.947,-177.631,6.561,148.504
C08113=1196.268,205.854,-58.971,-177.628,6.563,148.503
C08114=1196.264,206.102,-58.995,-177.626,6.565,148.503
C08115=1196.259,206.352,-59.020,-177.623,6.567,148.503
C08116=1196.255,206.600,-59.044,-177.621,6.569,148.503
C08117=1196.250,206.849,-59.068,-177.618,6.571,148.502
C08118=1196.245,207.098,-59.092,-177.615,6.573,148.502
C08119=1196.241,207.347,-59.117,-177.612,6.575,148.502
C08120=1196.237,207.595,-59.141,-177.610,6.577,148.501
C08121=1196.232,207.844,-59.166,-177.607,6.579,148.501
C08122=1196.227,208.093,-59.189,-177.605,6.581,148.501
C08123=1196.223,208.341,-59.213,-177.602,6.583,148.500
C08124=1196.218,208.591,-59.238,-177.600,6.585,148.500
C08125=1196.214,208.839,-59.262,-177.597,6.586,148.500
C08126=1196.209,209.088,-59.287,-177.594,6.589,148.499
C08127=1196.204,209.336,-59.311,-177.591,6.591,148.499
C08128=1196.200,209.586,-59.335,-177.589,6.593,148.499
C08129=1196.195,209.834,-59.360,-177.586,6.595,148.499
C08130=1196.191,210.083,-59.384,-177.584,6.597,148.498
C08131=1196.186,210.332,-59.409,-177.581,6.598,148.498
C08132=1196.182,210.603,-59.435,-177.578,6.601,148.498
C08133=1196.176,210.873,-59.461,-177.575,6.603,148.497
C08134=1196.171,211.143,-59.488,-177.572,6.605,148.497
C08135=1196.167,211.414,-59.515,-177.569,6.607,148.497
C08136=1196.162,211.662,-59.539,-177.567,6.610,148.497
C08137=1196.157,211.911,-59.564,-177.564,6.611,148.496
C08138=1196.153,212.159,-59.588,-177.562,6.613,148.496
C08139=1196.148,212.409,-59.613,-177.559,6.615,148.496
C08140=1196.144,212.657,-59.637,-177.556,6.618,148.495
C08141=1196.139,212.906,-59.662,-177.554,6.620,148.495
C08142=1196.135,213.155,-59.686,-177.551,6.622,148.495
C08143=1196.130,213.404,-59.711,-177.548,6.623,148.494
C08144=1196.125,213.652,-59.735,-177.546,6.625,148.494
C08145=1196.121,213.901,-59.761,-177.543,6.627,148.494
C08146=1196.116,214.150,-59.785,-177.540,6.630,148.494
C08147=1196.112,214.398,-59.809,-177.538,6.632,148.493
C08148=1196.107,214.647,-59.834,-177.535,6.634,148.493
C08149=1196.103,214.896,-59.858,-177.532,6.636,148.493
C08150=1196.098,215.145,-59.884,-177.530,6.638,148.493
C08151=1196.094,215.393,-59.908,-177.528,6.640,148.492
C08152=1196.089,215.642,-59.933,-177.524,6.642,148.492
C08153=1196.085,215.891,-59.957,-177.522,6.644,148.492
C08154=1196.080,216.140,-59.982,-177.520,6.646,148.492
C08155=1196.076,216.389,-60.007,-177.517,6.648,148.491
C08156=1196.071,216.637,-60.032,-177.514,6.650,148.491
C08157=1196.066,216.886,-60.057,-177.512,6.652,148.491
C08158=1196.062,217.135,-60.082,-177.508,6.654,148.490
C08159=1196.057,217.383,-60.106,-177.506,6.656,148.490
C08160=1196.053,217.632,-60.131,-177.504,6.658,148.490
C08161=1196.049,217.881,-60.156,-177.501,6.660,148.489
C08162=1196.044,218.129,-60.180,-177.498,6.662,148.489
C08163=1196.039,218.378,-60.206,-177.496,6.664,148.489
C08164=1196.035,218.627,-60.230,-177.493,6.667,148.489
C08165=1196.031,218.876,-60.255,-177.490,6.668,148.488
C08166=1196.026,219.124,-60.280,-177.488,6.670,148.488
C08167=1196.021,219.374,-60.305,-177.485,6.672,148.488
C08168=1196.017,219.621,-60.330,-177.483,6.674,148.488
C08169=1196.013,219.871,-60.355,-177.480,6.677,148.487
C08170=1196.007,220.120,-60.380,-177.477,6.679,148.487
C08171=1196.004,220.368,-60.405,-177.475,6.681,148.487
C08172=1195.999,220.617,-60.430,-177.472,6.683,148.487
C08173=1195.994,220.865,-60.455,-177.469,6.685,148.486
C08174=1195.989,221.114,-60.480,-177.467,6.688,148.486
C08175=1195.985,221.362,-60.505,-177.464,6.689,148.486
C08176=1195.981,221.611,-60.530,-177.461,6.691,148.485
C08177=1195.976,221.860,-60.555,-177.459,6.693,148.485
C08178=1195.971,222.109,-60.580,-177.457,6.695,148.485
C08179=1195.967,222.357,-60.605,-177.453,6.698,148.485
C08180=1195.963,222.606,-60.630,-177.451,6.700,148.484
C08181=1195.958,222.854,-60.656,-177.449,6.702,148.484
C08182=1195.954,223.104,-60.681,-177.446,6.704,148.484
C08183=1195.949,223.353,-60.706,-177.443,6.705,148.484
C08184=1195.944,223.601,-60.731,-177.441,6.708,148.484
C08185=1195.941,223.850,-60.756,-177.438,6.710,148.483
C08186=1195.936,224.098,-60.781,-177.435,6.712,148.483
C08187=1195.931,224.347,-60.807,-177.433,6.714,148.483
C08188=1195.926,224.595,-60.832,-177.431,6.716,148.482
C08189=1195.922,224.845,-60.857,-177.427,6.719,148.482
C08190=1195.917,225.093,-60.882,-177.425,6.721,148.482
C08191=1195.913,225.342,-60.908,-177.423,6.723,148.482
C08192=1195.909,225.590,-60.932,-177.420,6.725,148.481
C08193=1195.904,225.839,-60.958,-177.417,6.727,148.481
C08194=1195.900,226.088,-60.984,-177.414,6.729,148.481
C08195=1195.895,226.336,-61.008,-177.412,6.731,148.481
C08196=1195.891,226.585,-61.034,-177.409,6.733,148.480
C08197=1195.886,226.833,-61.060,-177.407,6.735,148.480
C08198=1195.881,227.083,-61.085,-177.404,6.738,148.480
C08199=1195.877,227.332,-61.110,-177.401,6.740,148.480
C08200=1195.872,227.580,-61.136,-177.399,6.742,148.479
C08201=1195.868,227.829,-61.162,-177.396,6.744,148.479
C08202=1195.863,228.077,-61.187,-177.393,6.746,148.479
C08203=1195.859,228.326,-61.212,-177.391,6.748,148.479
C08204=1195.854,228.575,-61.238,-177.388,6.750,148.478
C08205=1195.850,228.823,-61.263,-177.386,6.752,148.478
C08206=1195.845,229.072,-61.289,-177.383,6.755,148.478
C08207=1195.841,229.321,-61.315,-177.380,6.757,148.478
C08208=1195.836,229.569,-61.339,-177.378,6.759,148.477
C08209=1195.832,229.818,-61.365,-177.376,6.761,148.477
C08210=1195.828,230.067,-61.391,-177.372,6.764,148.477
C08211=1195.823,230.315,-61.416,-177.370,6.766,148.477
C08212=1195.819,230.564,-61.442,-177.368,6.768,148.477
C08213=1195.814,230.813,-61.468,-177.365,6.769,148.476
C08214=1195.810,231.061,-61.493,-177.362,6.772,148.476
C08215=1195.805,231.310,-61.519,-177.360,6.774,148.476
C08216=1195.801,231.558,-61.545,-177.357,6.776,148.476
C08217=1195.796,231.806,-61.570,-177.355,6.778,148.475
C08218=1195.792,232.055,-61.596,-177.352,6.781,148.475
C08219=1195.788,232.304,-61.621,-177.349,6.783,148.475
C08220=1195.782,232.552,-61.647,-177.347,6.785,148.475
C08221=1195.778,232.801,-61.673,-177.344,6.787,148.474
C08222=1195.774,233.050,-61.699,-177.341,6.790,148.474
C08223=1195.769,233.298,-61.724,-177.339,6.792,148.474
C08224=1195.765,233.547,-61.750,-177.336,6.793,148.474
C08225=1195.761,233.796,-61.776,-177.334,6.795,148.474
C08226=1195.756,234.045,-61.802,-177.331,6.798,148.473
C08227=1195.751,234.293,-61.828,-177.329,6.800,148.473
C08228=1195.746,234.542,-61.853,-177.326,6.802,148.473
C08229=1195.742,234.791,-61.879,-177.323,6.805,148.473
C08230=1195.738,235.039,-61.905,-177.321,6.807,148.472
C08231=1195.733,235.287,-61.930,-177.318,6.809,148.472
C08232=1195.729,235.536,-61.956,-177.316,6.811,148.472
C08233=1195.724,235.785,-61.982,-177.313,6.814,148.472
C08234=1195.720,236.034,-62.009,-177.310,6.815,148.471
C08235=1195.715,236.282,-62.034,-177.308,6.818,148.471
C08236=1195.711,236.554,-62.062,-177.305,6.820,148.471
C08237=1195.706,236.825,-62.091,-177.302,6.822,148.471
C08238=1195.701,237.097,-62.120,-177.299,6.825,148.471
C08239=1195.695,237.368,-62.147,-177.296,6.828,148.470
C08240=1195.692,237.616,-62.174,-177.293,6.830,148.470
C08241=1195.687,237.865,-62.199,-177.291,6.832,148.470
C08242=1195.682,238.114,-62.226,-177.289,6.834,148.470
C08243=1195.678,238.363,-62.252,-177.286,6.837,148.470
C08244=1195.674,238.611,-62.278,-177.283,6.838,148.469
C08245=1195.669,238.860,-62.304,-177.281,6.841,148.469
C08246=1195.664,239.109,-62.330,-177.278,6.843,148.469
C08247=1195.661,239.357,-62.356,-177.276,6.845,148.469
C08248=1195.656,239.606,-62.383,-177.273,6.847,148.468
C08249=1195.651,239.854,-62.408,-177.270,6.850,148.468
C08250=1195.647,240.102,-62.434,-177.268,6.852,148.468
C08251=1195.642,240.351,-62.461,-177.265,6.854,148.468
C08252=1195.638,240.600,-62.486,-177.262,6.857,148.468
C08253=1195.634,240.848,-62.513,-177.260,6.859,148.467
C08254=1195.629,241.097,-62.539,-177.258,6.861,148.467
C08255=1195.625,241.346,-62.565,-177.254,6.864,148.467
C08256=1195.620,241.594,-62.591,-177.252,6.866,148.467
C08257=1195.615,241.843,-62.618,-177.250,6.868,148.467
C08258=1195.611,242.091,-62.644,-177.247,6.870,148.466
C08259=1195.606,242.340,-62.670,-177.244,6.872,148.466
C08260=1195.602,242.588,-62.697,-177.242,6.875,148.466
C08261=1195.598,242.837,-62.723,-177.239,6.876,148.466
C08262=1195.593,243.086,-62.750,-177.237,6.879,148.466
C08263=1195.589,243.334,-62.775,-177.234,6.881,148.465
C08264=1195.584,243.583,-62.802,-177.232,6.883,148.465
C08265=1195.580,243.832,-62.828,-177.229,6.886,148.465
C08266=1195.576,244.080,-62.855,-177.226,6.888,148.465
C08267=1195.571,244.328,-62.881,-177.224,6.890,148.465
C08268=1195.566,244.577,-62.908,-177.221,6.893,148.464
C08269=1195.562,244.826,-62.933,-177.219,6.895,148.464
C08270=1195.557,245.074,-62.960,-177.215,6.898,148.464
C08271=1195.553,245.322,-62.987,-177.213,6.900,148.464
C08272=1195.548,245.571,-63.013,-177.211,6.902,148.464
C08273=1195.544,245.820,-63.040,-177.208,6.905,148.463
C08274=1195.539,246.069,-63.066,-177.206,6.907,148.463
C08275=1195.536,246.317,-63.093,-177.203,6.909,148.463
C08276=1195.531,246.565,-63.120,-177.200,6.912,148.463
C08277=1195.527,246.814,-63.145,-177.198,6.913,148.463
C08278=1195.522,247.063,-63.172,-177.195,6.916,148.463
C08279=1195.518,247.311,-63.199,-177.192,6.918,148.462
C08280=1195.513,247.560,-63.225,-177.190,6.920,148.462
C08281=1195.508,247.808,-63.252,-177.188,6.922,148.462
C08282=1195.505,248.057,-63.279,-177.185,6.925,148.462
C08283=1195.500,248.305,-63.306,-177.182,6.927,148.462
C08284=1195.496,248.554,-63.332,-177.179,6.930,148.461
C08285=1195.491,248.802,-63.359,-177.177,6.932,148.461
C08286=1195.486,249.051,-63.386,-177.175,6.934,148.461
C08287=1195.482,249.299,-63.412,-177.171,6.937,148.461
C08288=1195.477,249.548,-63.439,-177.169,6.939,148.461
C08289=1195.473,249.797,-63.466,-177.167,6.941,148.460
C08290=1195.469,250.045,-63.492,-177.164,6.944,148.460
C08291=1195.464,250.293,-63.519,-177.162,6.946,148.460
C08292=1195.460,250.542,-63.546,-177.159,6.949,148.460
C08293=1195.456,250.790,-63.573,-177.156,6.951,148.460
C08294=1195.451,251.039,-63.599,-177.154,6.953,148.460
C08295=1195.446,251.288,-63.626,-177.151,6.956,148.460
C08296=1195.442,251.536,-63.653,-177.148,6.957,148.459
C08297=1195.437,251.784,-63.680,-177.146,6.960,148.459
C08298=1195.433,252.034,-63.707,-177.143,6.962,148.459
C08299=1195.429,252.282,-63.734,-177.141,6.964,148.459
C08300=1195.425,252.530,-63.761,-177.138,6.967,148.459
C08301=1195.420,252.779,-63.788,-177.136,6.969,148.458
C08302=1195.416,253.027,-63.815,-177.133,6.972,148.458
C08303=1195.412,253.275,-63.841,-177.130,6.974,148.458
C08304=1195.407,253.524,-63.868,-177.128,6.976,148.458
C08305=1195.402,253.772,-63.895,-177.125,6.979,148.458
C08306=1195.398,254.021,-63.922,-177.123,6.981,148.458
C08307=1195.393,254.269,-63.949,-177.120,6.984,148.458
C08308=1195.390,254.518,-63.976,-177.117,6.986,148.457
C08309=1195.385,254.767,-64.003,-177.115,6.988,148.457
C08310=1195.380,255.015,-64.030,-177.112,6.991,148.457
C08311=1195.376,255.264,-64.057,-177.110,6.993,148.457
C08312=1195.371,255.512,-64.084,-177.107,6.996,148.457
C08313=1195.367,255.760,-64.111,-177.105,6.998,148.456
C08314=1195.362,256.009,-64.138,-177.102,7.000,148.456
C08315=1195.358,256.258,-64.165,-177.099,7.003,148.456
C08316=1195.354,256.507,-64.192,-177.097,7.005,148.456
C08317=1195.349,256.755,-64.220,-177.094,7.008,148.456
C08318=1195.345,257.003,-64.247,-177.092,7.010,148.456
C08319=1195.340,257.252,-64.274,-177.089,7.013,148.456
C08320=1195.335,257.500,-64.301,-177.087,7.015,148.455
C08321=1195.332,257.749,-64.328,-177.084,7.017,148.455
C08322=1195.328,257.997,-64.356,-177.081,7.020,148.455
C08323=1195.323,258.245,-64.383,-177.079,7.021,148.455
C08324=1195.318,258.494,-64.410,-177.076,7.024,148.455
C08325=1195.314,258.742,-64.437,-177.074,7.027,148.455
C08326=1195.310,258.992,-64.465,-177.071,7.029,148.454
C08327=1195.305,259.239,-64.492,-177.069,7.031,148.454
C08328=1195.301,259.488,-64.519,-177.066,7.034,148.454
C08329=1195.296,259.736,-64.547,-177.063,7.036,148.454
C08330=1195.292,259.985,-64.575,-177.061,7.038,148.454
C08331=1195.288,260.233,-64.602,-177.058,7.041,148.454
C08332=1195.283,260.482,-64.629,-177.056,7.043,148.453
C08333=1195.279,260.730,-64.657,-177.053,7.046,148.453
C08334=1195.275,260.979,-64.684,-177.050,7.048,148.453
C08335=1195.270,261.228,-64.711,-177.048,7.051,148.453
C08336=1195.266,261.475,-64.739,-177.046,7.053,148.453
C08337=1195.261,261.724,-64.766,-177.042,7.056,148.453
C08338=1195.257,261.973,-64.793,-177.040,7.058,148.453
C08339=1195.253,262.221,-64.821,-177.038,7.061,148.453
C08340=1195.247,262.494,-64.851,-177.035,7.063,148.452
C08341=1195.243,262.767,-64.882,-177.032,7.066,148.452
C08342=1195.238,263.039,-64.912,-177.029,7.069,148.452
C08343=1195.233,263.312,-64.942,-177.026,7.072,148.452
C08344=1195.229,263.561,-64.970,-177.024,7.074,148.452
C08345=1195.224,263.809,-64.997,-177.021,7.077,148.452
C08346=1195.220,264.057,-65.024,-177.019,7.079,148.452
C08347=1195.216,264.306,-65.053,-177.016,7.082,148.451
C08348=1195.211,264.554,-65.080,-177.013,7.084,148.451
C08349=1195.207,264.802,-65.107,-177.011,7.087,148.451
C08350=1195.203,265.052,-65.135,-177.009,7.089,148.451
C08351=1195.198,265.300,-65.163,-177.005,7.091,148.451
C08352=1195.193,265.548,-65.190,-177.003,7.094,148.451
C08353=1195.189,265.797,-65.218,-177.001,7.097,148.451
C08354=1195.185,266.045,-65.245,-176.998,7.098,148.450
C08355=1195.180,266.293,-65.273,-176.995,7.101,148.450
C08356=1195.177,266.542,-65.301,-176.993,7.104,148.450
C08357=1195.171,266.791,-65.329,-176.990,7.107,148.450
C08358=1195.167,267.038,-65.357,-176.988,7.108,148.450
C08359=1195.163,267.287,-65.385,-176.985,7.111,148.450
C08360=1195.159,267.536,-65.412,-176.983,7.114,148.450
C08361=1195.153,267.784,-65.440,-176.980,7.116,148.449
C08362=1195.150,268.032,-65.469,-176.978,7.118,148.449
C08363=1195.145,268.281,-65.496,-176.975,7.121,148.449
C08364=1195.141,268.529,-65.524,-176.973,7.124,148.449
C08365=1195.137,268.777,-65.552,-176.969,7.126,148.449
C08366=1195.132,269.026,-65.579,-176.967,7.128,148.449
C08367=1195.128,269.275,-65.607,-176.965,7.131,148.449
C08368=1195.123,269.522,-65.635,-176.962,7.133,148.449
C08369=1195.119,269.771,-65.664,-176.959,7.136,148.449
C08370=1195.115,270.019,-65.692,-176.957,7.139,148.448
C08371=1195.111,270.268,-65.719,-176.954,7.142,148.448
C08372=1195.106,270.516,-65.747,-176.952,7.143,148.448
C08373=1195.101,270.764,-65.775,-176.949,7.146,148.448
C08374=1195.097,271.013,-65.803,-176.947,7.149,148.448
C08375=1195.093,271.261,-65.831,-176.944,7.152,148.448
C08376=1195.089,271.510,-65.860,-176.941,7.154,148.448
C08377=1195.084,271.758,-65.887,-176.939,7.156,148.448
C08378=1195.079,272.007,-65.916,-176.936,7.159,148.448
C08379=1195.075,272.255,-65.943,-176.934,7.162,148.448
C08380=1195.071,272.504,-65.972,-176.931,7.164,148.447
C08381=1195.066,272.752,-66.000,-176.929,7.166,148.447
C08382=1195.062,273.000,-66.028,-176.926,7.169,148.447
C08383=1195.058,273.248,-66.056,-176.924,7.172,148.447
C08384=1195.054,273.497,-66.085,-176.921,7.174,148.447
C08385=1195.049,273.745,-66.112,-176.918,7.176,148.447
C08386=1195.045,273.994,-66.141,-176.916,7.179,148.447
C08387=1195.040,274.242,-66.169,-176.914,7.182,148.447
C08388=1195.037,274.490,-66.197,-176.911,7.185,148.447
C08389=1195.032,274.739,-66.225,-176.908,7.187,148.446
C08390=1195.028,274.987,-66.254,-176.906,7.189,148.446
C08391=1195.023,275.235,-66.282,-176.903,7.192,148.446
C08392=1195.019,275.484,-66.310,-176.901,7.195,148.446
C08393=1195.014,275.732,-66.338,-176.898,7.198,148.446
C08394=1195.010,275.981,-66.367,-176.895,7.200,148.446
C08395=1195.005,276.229,-66.395,-176.893,7.203,148.446
C08396=1195.001,276.477,-66.423,-176.890,7.206,148.446
C08397=1194.997,276.725,-66.452,-176.888,7.208,148.446
C08398=1194.993,276.974,-66.480,-176.885,7.211,148.446
C08399=1194.988,277.222,-66.509,-176.883,7.213,148.445
C08400=1194.984,277.470,-66.537,-176.880,7.216,148.445
C08401=1194.979,277.719,-66.566,-176.878,7.218,148.445
C08402=1194.975,277.967,-66.593,-176.875,7.221,148.445
C08403=1194.971,278.215,-66.623,-176.872,7.224,148.445
C08404=1194.967,278.464,-66.651,-176.870,7.226,148.445
C08405=1194.962,278.712,-66.679,-176.867,7.229,148.445
C08406=1194.958,278.961,-66.708,-176.865,7.231,148.445
C08407=1194.953,279.209,-66.736,-176.862,7.234,148.445
C08408=1194.949,279.457,-66.765,-176.860,7.236,148.445
C08409=1194.945,279.706,-66.793,-176.857,7.239,148.445
C08410=1194.940,279.954,-66.822,-176.854,7.242,148.444
C08411=1194.936,280.202,-66.851,-176.852,7.244,148.444
C08412=1194.932,280.450,-66.879,-176.849,7.247,148.444
C08413=1194.927,280.699,-66.908,-176.847,7.249,148.444
C08414=1194.923,280.947,-66.937,-176.844,7.252,148.444
C08415=1194.919,281.195,-66.965,-176.842,7.255,148.444
C08416=1194.914,281.444,-66.994,-176.839,7.257,148.444
C08417=1194.911,281.692,-67.023,-176.836,7.260,148.444
C08418=1194.906,281.940,-67.051,-176.834,7.262,148.444
C08419=1194.901,282.189,-67.080,-176.831,7.265,148.444
C08420=1194.897,282.437,-67.109,-176.829,7.268,148.444
C08421=1194.893,282.685,-67.137,-176.827,7.270,148.444
C08422=1194.888,282.933,-67.166,-176.824,7.273,148.444
C08423=1194.884,283.182,-67.195,-176.821,7.275,148.443
C08424=1194.880,283.430,-67.224,-176.819,7.278,148.443
C08425=1194.875,283.678,-67.252,-176.816,7.281,148.443
C08426=1194.871,283.927,-67.282,-176.814,7.283,148.443
C08427=1194.866,284.175,-67.310,-176.811,7.286,148.443
C08428=1194.863,284.423,-67.339,-176.809,7.288,148.443
C08429=1194.858,284.672,-67.368,-176.806,7.291,148.443
C08430=1194.854,284.920,-67.397,-176.803,7.294,148.443
C08431=1194.849,285.168,-67.426,-176.801,7.297,148.443
C08432=1194.845,285.417,-67.455,-176.798,7.299,148.443
C08433=1194.841,285.665,-67.483,-176.795,7.302,148.443
C08434=1194.837,285.913,-67.513,-176.793,7.305,148.442
C08435=1194.832,286.162,-67.541,-176.791,7.308,148.442
C08436=1194.828,286.410,-67.570,-176.788,7.310,148.442
C08437=1194.823,286.658,-67.600,-176.786,7.313,148.442
C08438=1194.819,286.907,-67.629,-176.783,7.316,148.442
C08439=1194.815,287.154,-67.657,-176.781,7.318,148.442
C08440=1194.811,287.402,-67.687,-176.778,7.321,148.442
C08441=1194.806,287.651,-67.715,-176.775,7.324,148.442
C08442=1194.802,287.900,-67.745,-176.773,7.326,148.442
C08443=1194.797,288.147,-67.774,-176.770,7.329,148.442
C08444=1194.793,288.422,-67.806,-176.767,7.332,148.442
C08445=1194.788,288.697,-67.838,-176.765,7.335,148.442
C08446=1194.783,288.971,-67.870,-176.762,7.338,148.442
C08447=1194.779,289.246,-67.902,-176.759,7.341,148.442
C08448=1194.774,289.493,-67.932,-176.757,7.344,148.442
C08449=1194.770,289.742,-67.961,-176.754,7.346,148.442
C08450=1194.765,289.990,-67.990,-176.752,7.349,148.442
C08451=1194.761,290.239,-68.019,-176.749,7.352,148.441
C08452=1194.757,290.487,-68.049,-176.746,7.354,148.441
C08453=1194.752,290.735,-68.078,-176.744,7.357,148.441
C08454=1194.748,290.983,-68.107,-176.742,7.359,148.441
C08455=1194.744,291.232,-68.136,-176.739,7.362,148.441
C08456=1194.739,291.480,-68.165,-176.736,7.365,148.441
C08457=1194.735,291.728,-68.195,-176.734,7.367,148.441
C08458=1194.731,291.977,-68.224,-176.731,7.370,148.441
C08459=1194.727,292.225,-68.254,-176.729,7.373,148.441
C08460=1194.722,292.472,-68.283,-176.726,7.375,148.441
C08461=1194.718,292.721,-68.312,-176.724,7.378,148.441
C08462=1194.714,292.969,-68.342,-176.721,7.381,148.441
C08463=1194.709,293.217,-68.371,-176.719,7.384,148.441
C08464=1194.705,293.465,-68.401,-176.716,7.387,148.441
C08465=1194.701,293.714,-68.430,-176.713,7.390,148.441
C08466=1194.697,293.962,-68.460,-176.711,7.392,148.441
C08467=1194.693,294.210,-68.489,-176.709,7.395,148.441
C08468=1194.689,294.458,-68.518,-176.706,7.398,148.441
C08469=1194.684,294.707,-68.548,-176.704,7.400,148.441
C08470=1194.680,294.954,-68.577,-176.701,7.403,148.441
C08471=1194.675,295.203,-68.606,-176.698,7.406,148.441
C08472=1194.670,295.451,-68.637,-176.696,7.408,148.441
C08473=1194.666,295.699,-68.666,-176.693,7.411,148.441
C08474=1194.662,295.948,-68.695,-176.691,7.414,148.441
C08475=1194.658,296.196,-68.725,-176.688,7.417,148.440
C08476=1194.654,296.444,-68.754,-176.686,7.419,148.440
C08477=1194.650,296.693,-68.784,-176.683,7.422,148.440
C08478=1194.646,296.940,-68.814,-176.681,7.425,148.440
C08479=1194.641,297.189,-68.844,-176.678,7.428,148.440
C08480=1194.637,297.437,-68.873,-176.676,7.431,148.440
C08481=1194.632,297.685,-68.903,-176.673,7.434,148.440
C08482=1194.628,297.934,-68.932,-176.671,7.436,148.440
C08483=1194.624,298.182,-68.962,-176.668,7.439,148.440
C08484=1194.619,298.430,-68.993,-176.665,7.442,148.440
C08485=1194.615,298.678,-69.022,-176.663,7.444,148.440
C08486=1194.611,298.926,-69.051,-176.661,7.447,148.440
C08487=1194.607,299.175,-69.081,-176.658,7.450,148.440
C08488=1194.602,299.423,-69.112,-176.655,7.453,148.440
C08489=1194.598,299.671,-69.141,-176.653,7.456,148.440
C08490=1194.594,299.919,-69.171,-176.651,7.459,148.440
C08491=1194.590,300.167,-69.201,-176.648,7.462,148.440
C08492=1194.585,300.415,-69.231,-176.646,7.464,148.440
C08493=1194.581,300.664,-69.260,-176.643,7.467,148.440
C08494=1194.577,300.911,-69.290,-176.641,7.470,148.440
C08495=1194.573,301.159,-69.320,-176.638,7.472,148.440
C08496=1194.568,301.408,-69.350,-176.636,7.475,148.440
C08497=1194.564,301.656,-69.380,-176.633,7.478,148.440
C08498=1194.560,301.904,-69.410,-176.630,7.481,148.440
C08499=1194.555,302.153,-69.440,-176.628,7.483,148.440
C08500=1194.551,302.400,-69.470,-176.625,7.486,148.440
C08501=1194.547,302.648,-69.499,-176.623,7.489,148.440
C08502=1194.542,302.896,-69.530,-176.621,7.492,148.440
C08503=1194.539,303.145,-69.560,-176.618,7.495,148.440
C08504=1194.534,303.393,-69.591,-176.616,7.498,148.440
C08505=1194.530,303.642,-69.620,-176.613,7.501,148.440
C08506=1194.526,303.889,-69.650,-176.611,7.503,148.440
C08507=1194.521,304.138,-69.680,-176.608,7.506,148.440
C08508=1194.517,304.385,-69.710,-176.605,7.509,148.440
C08509=1194.512,304.634,-69.740,-176.603,7.511,148.440
C08510=1194.508,304.882,-69.771,-176.601,7.514,148.440
C08511=1194.504,305.130,-69.801,-176.598,7.518,148.440
C08512=1194.500,305.378,-69.831,-176.596,7.521,148.440
C08513=1194.496,305.626,-69.860,-176.593,7.523,148.440
C08514=1194.492,305.875,-69.891,-176.591,7.526,148.440
C08515=1194.488,306.122,-69.922,-176.588,7.529,148.440
C08516=1194.483,306.371,-69.952,-176.585,7.532,148.440
C08517=1194.479,306.619,-69.982,-176.583,7.534,148.440
C08518=1194.474,306.867,-70.012,-176.581,7.537,148.440
C08519=1194.470,307.115,-70.042,-176.578,7.540,148.440
C08520=1194.465,307.363,-70.073,-176.576,7.542,148.440
C08521=1194.462,307.612,-70.103,-176.573,7.545,148.440
C08522=1194.457,307.860,-70.133,-176.571,7.548,148.440
C08523=1194.453,308.108,-70.164,-176.568,7.551,148.440
C08524=1194.449,308.355,-70.194,-176.566,7.554,148.440
C08525=1194.444,308.604,-70.224,-176.564,7.557,148.440
C08526=1194.441,308.852,-70.255,-176.561,7.560,148.440
C08527=1194.436,309.100,-70.286,-176.558,7.563,148.440
C08528=1194.432,309.348,-70.316,-176.556,7.565,148.440
C08529=1194.427,309.597,-70.346,-176.554,7.569,148.440
C08530=1194.423,309.844,-70.376,-176.551,7.572,148.440
C08531=1194.419,310.093,-70.407,-176.548,7.575,148.440
C08532=1194.415,310.341,-70.438,-176.546,7.577,148.440
C08533=1194.411,310.588,-70.468,-176.544,7.580,148.440
C08534=1194.406,310.837,-70.498,-176.541,7.583,148.440
C08535=1194.401,311.085,-70.529,-176.539,7.586,148.440
C08536=1194.398,311.333,-70.559,-176.537,7.588,148.440
C08537=1194.393,311.581,-70.590,-176.534,7.591,148.440
C08538=1194.389,311.829,-70.621,-176.531,7.594,148.440
C08539=1194.385,312.077,-70.651,-176.529,7.598,148.440
C08540=1194.381,312.326,-70.682,-176.527,7.600,148.440
C08541=1194.376,312.574,-70.713,-176.524,7.603,148.440
C08542=1194.372,312.821,-70.743,-176.521,7.606,148.440
C08543=1194.368,313.069,-70.774,-176.519,7.609,148.440
C08544=1194.364,313.318,-70.805,-176.517,7.611,148.440
C08545=1194.360,313.565,-70.835,-176.514,7.614,148.440
C08546=1194.355,313.813,-70.866,-176.512,7.617,148.440
C08547=1194.351,314.062,-70.897,-176.509,7.621,148.441
C08548=1194.346,314.338,-70.931,-176.507,7.624,148.441
C08549=1194.342,314.615,-70.965,-176.504,7.627,148.441
C08550=1194.337,314.891,-71.000,-176.501,7.630,148.441
C08551=1194.332,315.167,-71.033,-176.499,7.633,148.441
C08552=1194.328,315.416,-71.064,-176.496,7.636,148.441
C08553=1194.323,315.664,-71.095,-176.494,7.639,148.441
C08554=1194.319,315.912,-71.126,-176.491,7.642,148.441
C08555=1194.316,316.159,-71.157,-176.489,7.645,148.441
C08556=1194.311,316.407,-71.188,-176.487,7.648,148.441
C08557=1194.307,316.655,-71.219,-176.484,7.651,148.441
C08558=1194.303,316.904,-71.250,-176.482,7.654,148.441
C08559=1194.298,317.152,-71.281,-176.479,7.657,148.441
C08560=1194.294,317.401,-71.312,-176.477,7.659,148.441
C08561=1194.290,317.648,-71.343,-176.475,7.663,148.441
C08562=1194.286,317.896,-71.373,-176.472,7.666,148.441
C08563=1194.282,318.144,-71.404,-176.469,7.669,148.441
C08564=1194.277,318.392,-71.435,-176.468,7.671,148.441
C08565=1194.273,318.640,-71.466,-176.465,7.674,148.441
C08566=1194.269,318.888,-71.498,-176.462,7.677,148.441
C08567=1194.264,319.136,-71.529,-176.460,7.680,148.442
C08568=1194.261,319.385,-71.559,-176.458,7.683,148.442
C08569=1194.257,319.632,-71.591,-176.455,7.686,148.442
C08570=1194.252,319.880,-71.621,-176.453,7.689,148.442
C08571=1194.248,320.129,-71.653,-176.450,7.692,148.442
C08572=1194.244,320.376,-71.684,-176.447,7.695,148.442
C08573=1194.240,320.625,-71.715,-176.446,7.697,148.442
C08574=1194.235,320.872,-71.746,-176.443,7.701,148.442
C08575=1194.231,321.121,-71.778,-176.441,7.704,148.442
C08576=1194.227,321.368,-71.809,-176.438,7.707,148.442
C08577=1194.222,321.616,-71.839,-176.436,7.709,148.442
C08578=1194.219,321.864,-71.871,-176.434,7.712,148.442
C08579=1194.214,322.112,-71.902,-176.431,7.715,148.442
C08580=1194.210,322.360,-71.934,-176.429,7.719,148.442
C08581=1194.206,322.608,-71.964,-176.426,7.722,148.442
C08582=1194.202,322.856,-71.996,-176.424,7.724,148.442
C08583=1194.197,323.104,-72.027,-176.422,7.727,148.443
C08584=1194.194,323.352,-72.059,-176.419,7.730,148.443
C08585=1194.189,323.600,-72.090,-176.417,7.734,148.443
C08586=1194.185,323.848,-72.122,-176.414,7.737,148.443
C08587=1194.181,324.096,-72.152,-176.412,7.739,148.443
C08588=1194.177,324.344,-72.184,-176.410,7.742,148.443
C08589=1194.172,324.592,-72.215,-176.407,7.745,148.443
C08590=1194.169,324.840,-72.247,-176.405,7.748,148.443
C08591=1194.164,325.088,-72.278,-176.403,7.751,148.443
C08592=1194.160,325.336,-72.309,-176.400,7.754,148.443
C08593=1194.156,325.584,-72.341,-176.398,7.757,148.443
C08594=1194.152,325.832,-72.372,-176.395,7.760,148.444
C08595=1194.147,326.080,-72.404,-176.393,7.763,148.444
C08596=1194.143,326.329,-72.435,-176.391,7.766,148.444
C08597=1194.139,326.576,-72.467,-176.388,7.769,148.444
C08598=1194.135,326.824,-72.499,-176.386,7.772,148.444
C08599=1194.131,327.073,-72.530,-176.383,7.775,148.444
C08600=1194.127,327.320,-72.561,-176.381,7.779,148.444
C08601=1194.123,327.568,-72.593,-176.379,7.781,148.444
C08602=1194.118,327.816,-72.625,-176.377,7.784,148.444
C08603=1194.114,328.064,-72.656,-176.374,7.787,148.444
C08604=1194.109,328.312,-72.688,-176.372,7.790,148.445
C08605=1194.106,328.560,-72.719,-176.370,7.794,148.445
C08606=1194.101,328.807,-72.751,-176.368,7.796,148.445
C08607=1194.097,329.056,-72.783,-176.365,7.799,148.445
C08608=1194.093,329.304,-72.815,-176.363,7.802,148.445
C08609=1194.089,329.552,-72.846,-176.360,7.806,148.445
C08610=1194.085,329.800,-72.878,-176.358,7.809,148.445
C08611=1194.080,330.047,-72.910,-176.356,7.811,148.445
C08612=1194.076,330.296,-72.941,-176.353,7.814,148.445
C08613=1194.072,330.544,-72.973,-176.351,7.817,148.446
C08614=1194.068,330.791,-73.004,-176.349,7.821,148.446
C08615=1194.063,331.040,-73.037,-176.346,7.824,148.446
C08616=1194.060,331.288,-73.069,-176.344,7.826,148.446
C08617=1194.055,331.535,-73.100,-176.342,7.829,148.446
C08618=1194.051,331.783,-73.133,-176.340,7.833,148.446
C08619=1194.047,332.031,-73.164,-176.337,7.836,148.446
C08620=1194.043,332.279,-73.196,-176.335,7.839,148.446
C08621=1194.039,332.527,-73.227,-176.333,7.841,148.446
C08622=1194.034,332.775,-73.259,-176.331,7.845,148.447
C08623=1194.030,333.023,-73.291,-176.328,7.848,148.447
C08624=1194.026,333.271,-73.323,-176.326,7.851,148.447
C08625=1194.022,333.519,-73.355,-176.324,7.854,148.447
C08626=1194.018,333.767,-73.387,-176.321,7.857,148.447
C08627=1194.013,334.015,-73.419,-176.319,7.860,148.447
C08628=1194.009,334.262,-73.451,-176.317,7.863,148.448
C08629=1194.006,334.510,-73.483,-176.314,7.866,148.448
C08630=1194.001,334.758,-73.516,-176.312,7.870,148.448
C08631=1193.997,335.006,-73.548,-176.310,7.872,148.448
C08632=1193.992,335.254,-73.580,-176.308,7.875,148.448
C08633=1193.989,335.502,-73.611,-176.305,7.879,148.448
C08634=1193.985,335.750,-73.643,-176.303,7.882,148.448
C08635=1193.980,335.998,-73.675,-176.300,7.885,148.448
C08636=1193.976,336.246,-73.707,-176.299,7.887,148.449
C08637=1193.972,336.494,-73.740,-176.297,7.891,148.449
C08638=1193.968,336.741,-73.772,-176.294,7.894,148.449
C08639=1193.963,336.989,-73.804,-176.292,7.897,148.449
C08640=1193.960,337.237,-73.836,-176.289,7.900,148.449
C08641=1193.955,337.486,-73.869,-176.288,7.903,148.449
C08642=1193.952,337.734,-73.900,-176.285,7.906,148.450
C08643=1193.947,337.981,-73.933,-176.283,7.909,148.450
C08644=1193.943,338.229,-73.965,-176.281,7.913,148.450
C08645=1193.939,338.477,-73.997,-176.278,7.916,148.450
C08646=1193.935,338.725,-74.029,-176.276,7.919,148.450
C08647=1193.930,338.972,-74.062,-176.274,7.922,148.450
C08648=1193.927,339.220,-74.094,-176.272,7.925,148.450
C08649=1193.922,339.468,-74.126,-176.269,7.928,148.451
C08650=1193.919,339.716,-74.159,-176.267,7.931,148.451
C08651=1193.914,339.964,-74.191,-176.265,7.935,148.451
C08652=1193.909,340.242,-74.228,-176.263,7.938,148.451
C08653=1193.904,340.521,-74.263,-176.260,7.941,148.451
C08654=1193.900,340.800,-74.300,-176.258,7.944,148.451
C08655=1193.895,341.078,-74.337,-176.255,7.949,148.452
C08656=1193.891,341.327,-74.369,-176.253,7.951,148.452
C08657=1193.888,341.574,-74.402,-176.251,7.954,148.452
C08658=1193.883,341.822,-74.434,-176.249,7.958,148.452
C08659=1193.878,342.069,-74.467,-176.247,7.961,148.453
C08660=1193.875,342.318,-74.499,-176.244,7.964,148.453
C08661=1193.871,342.565,-74.532,-176.242,7.967,148.453
C08662=1193.866,342.814,-74.564,-176.240,7.970,148.453
C08663=1193.863,343.061,-74.597,-176.238,7.973,148.453
C08664=1193.858,343.309,-74.629,-176.236,7.977,148.453
C08665=1193.854,343.556,-74.662,-176.233,7.980,148.454
C08666=1193.850,343.804,-74.694,-176.231,7.983,148.454
C08667=1193.846,344.052,-74.727,-176.229,7.986,148.454
C08668=1193.841,344.301,-74.759,-176.227,7.989,148.454
C08669=1193.838,344.548,-74.792,-176.225,7.992,148.454
C08670=1193.833,344.796,-74.824,-176.223,7.996,148.455
C08671=1193.829,345.043,-74.857,-176.220,7.999,148.455
C08672=1193.824,345.292,-74.890,-176.219,8.002,148.455
C08673=1193.821,345.539,-74.922,-176.217,8.005,148.455
C08674=1193.817,345.787,-74.955,-176.214,8.008,148.456
C08675=1193.812,346.035,-74.988,-176.212,8.012,148.456
C08676=1193.808,346.283,-75.021,-176.210,8.015,148.456
C08677=1193.805,346.530,-75.054,-176.208,8.017,148.456
C08678=1193.800,346.779,-75.086,-176.206,8.021,148.456
C08679=1193.796,347.026,-75.119,-176.204,8.024,148.457
C08680=1193.792,347.274,-75.152,-176.201,8.027,148.457
C08681=1193.788,347.522,-75.185,-176.199,8.031,148.457
C08682=1193.784,347.770,-75.217,-176.197,8.034,148.457
C08683=1193.779,348.017,-75.250,-176.195,8.036,148.457
C08684=1193.775,348.265,-75.283,-176.193,8.040,148.458
C08685=1193.771,348.513,-75.316,-176.191,8.043,148.458
C08686=1193.767,348.761,-75.349,-176.189,8.046,148.458
C08687=1193.763,349.008,-75.382,-176.187,8.050,148.459
C08688=1193.758,349.256,-75.415,-176.185,8.053,148.459
C08689=1193.755,349.504,-75.447,-176.183,8.056,148.459
C08690=1193.751,349.752,-75.480,-176.181,8.059,148.459
C08691=1193.746,350.000,-75.513,-176.178,8.063,148.459
C08692=1193.742,350.247,-75.547,-176.176,8.066,148.460
C08693=1193.738,350.495,-75.580,-176.174,8.068,148.460
C08694=1193.734,350.743,-75.612,-176.173,8.072,148.460
C08695=1193.730,350.991,-75.645,-176.170,8.075,148.460
C08696=1193.725,351.239,-75.678,-176.168,8.079,148.461
C08697=1193.721,351.487,-75.712,-176.166,8.082,148.461
C08698=1193.717,351.734,-75.745,-176.164,8.085,148.461
C08699=1193.714,351.982,-75.777,-176.162,8.088,148.461
C08700=1193.710,352.230,-75.810,-176.160,8.091,148.462
C08701=1193.706,352.477,-75.844,-176.158,8.095,148.462
C08702=1193.701,352.725,-75.877,-176.156,8.098,148.462
C08703=1193.697,352.973,-75.910,-176.154,8.101,148.462
C08704=1193.693,353.220,-75.943,-176.152,8.104,148.463
C08705=1193.689,353.468,-75.976,-176.150,8.108,148.463
C08706=1193.685,353.716,-76.009,-176.148,8.111,148.463
C08707=1193.681,353.964,-76.043,-176.146,8.115,148.464
C08708=1193.677,354.212,-76.076,-176.144,8.117,148.464
C08709=1193.673,354.460,-76.109,-176.142,8.120,148.464
C08710=1193.669,354.708,-76.142,-176.140,8.124,148.464
C08711=1193.665,354.955,-76.176,-176.138,8.127,148.465
C08712=1193.661,355.203,-76.209,-176.136,8.131,148.465
C08713=1193.656,355.451,-76.242,-176.135,8.133,148.465
C08714=1193.652,355.698,-76.275,-176.132,8.137,148.466
C08715=1193.647,355.946,-76.309,-176.130,8.140,148.466
C08716=1193.644,356.194,-76.343,-176.128,8.144,148.466
C08717=1193.639,356.441,-76.376,-176.126,8.147,148.466
C08718=1193.635,356.689,-76.409,-176.124,8.150,148.467
C08719=1193.631,356.937,-76.442,-176.123,8.153,148.467
C08720=1193.628,357.185,-76.476,-176.120,8.157,148.467
C08721=1193.624,357.433,-76.509,-176.119,8.160,148.468
C08722=1193.620,357.680,-76.543,-176.116,8.164,148.468
C08723=1193.616,357.928,-76.576,-176.115,8.166,148.468
C08724=1193.611,358.176,-76.609,-176.113,8.170,148.469
C08725=1193.607,358.423,-76.642,-176.111,8.173,148.469
C08726=1193.602,358.671,-76.676,-176.109,8.177,148.469
C08727=1193.599,358.919,-76.710,-176.107,8.180,148.469
C08728=1193.595,359.167,-76.743,-176.105,8.183,148.470
C08729=1193.591,359.415,-76.776,-176.103,8.186,148.470
C08730=1193.587,359.662,-76.810,-176.101,8.190,148.470
C08731=1193.583,359.909,-76.843,-176.100,8.193,148.471
C08732=1193.578,360.157,-76.877,-176.098,8.196,148.471
C08733=1193.575,360.405,-76.911,-176.096,8.199,148.472
C08734=1193.571,360.653,-76.945,-176.094,8.203,148.472
C08735=1193.567,360.901,-76.978,-176.092,8.206,148.472
C08736=1193.563,361.148,-77.012,-176.091,8.209,148.473
C08737=1193.558,361.396,-77.045,-176.089,8.213,148.473
C08738=1193.554,361.644,-77.079,-176.087,8.216,148.473
C08739=1193.550,361.891,-77.113,-176.085,8.220,148.473
C08740=1193.546,362.139,-77.146,-176.083,8.222,148.474
C08741=1193.542,362.386,-77.180,-176.082,8.226,148.474
C08742=1193.538,362.634,-77.214,-176.080,8.230,148.475
C08743=1193.534,362.883,-77.247,-176.078,8.232,148.475
C08744=1193.530,363.130,-77.281,-176.076,8.236,148.475
C08745=1193.525,363.378,-77.315,-176.075,8.239,148.476
C08746=1193.522,363.625,-77.349,-176.073,8.242,148.476
C08747=1193.517,363.873,-77.382,-176.071,8.246,148.476
C08748=1193.514,364.120,-77.416,-176.069,8.249,148.477
C08749=1193.509,364.369,-77.450,-176.068,8.252,148.477
C08750=1193.505,364.616,-77.484,-176.066,8.256,148.478
C08751=1193.501,364.863,-77.517,-176.064,8.259,148.478
C08752=1193.497,365.111,-77.552,-176.063,8.262,148.478
C08753=1193.494,365.359,-77.585,-176.061,8.265,148.479
C08754=1193.489,365.606,-77.619,-176.059,8.269,148.479
C08755=1193.485,365.854,-77.653,-176.058,8.272,148.480
C08756=1193.481,366.135,-77.692,-176.056,8.275,148.480
C08757=1193.476,366.416,-77.730,-176.054,8.279,148.480
C08758=1193.471,366.698,-77.769,-176.052,8.283,148.481
C08759=1193.467,366.978,-77.807,-176.050,8.287,148.481
C08760=1193.463,367.225,-77.841,-176.049,8.290,148.482
C08761=1193.459,367.474,-77.874,-176.047,8.294,148.482
C08762=1193.455,367.721,-77.909,-176.046,8.296,148.483
C08763=1193.451,367.968,-77.943,-176.044,8.300,148.483
C08764=1193.446,368.216,-77.977,-176.042,8.304,148.483
C08765=1193.443,368.464,-78.011,-176.041,8.306,148.484
C08766=1193.439,368.711,-78.045,-176.039,8.310,148.484
C08767=1193.434,368.959,-78.078,-176.038,8.313,148.485
C08768=1193.431,369.207,-78.113,-176.036,8.316,148.485
C08769=1193.426,369.455,-78.147,-176.035,8.319,148.485
C08770=1193.423,369.702,-78.181,-176.033,8.323,148.486
C08771=1193.418,369.950,-78.215,-176.032,8.326,148.486
C08772=1193.414,370.197,-78.249,-176.030,8.329,148.487
C08773=1193.410,370.445,-78.283,-176.029,8.332,148.487
C08774=1193.407,370.693,-78.318,-176.027,8.336,148.488
C08775=1193.402,370.941,-78.351,-176.027,8.339,148.488
C08776=1193.398,371.188,-78.385,-176.025,8.343,148.489
C08777=1193.394,371.436,-78.420,-176.024,8.345,148.489
C08778=1193.390,371.683,-78.454,-176.022,8.349,148.489
C08779=1193.386,371.931,-78.488,-176.020,8.352,148.490
C08780=1193.382,372.178,-78.523,-176.019,8.355,148.490
C08781=1193.377,372.426,-78.556,-176.018,8.358,148.491
C08782=1193.374,372.674,-78.591,-176.017,8.361,148.491
C08783=1193.370,372.922,-78.625,-176.015,8.365,148.492
C08784=1193.366,373.169,-78.659,-176.014,8.368,148.492
C08785=1193.362,373.417,-78.694,-176.012,8.372,148.493
C08786=1193.358,373.664,-78.728,-176.011,8.374,148.493
C08787=1193.353,373.911,-78.762,-176.010,8.377,148.493
C08788=1193.350,374.159,-78.796,-176.009,8.381,148.494
C08789=1193.346,374.407,-78.831,-176.007,8.384,148.494
C08790=1193.342,374.655,-78.866,-176.006,8.387,148.495
C08791=1193.338,374.902,-78.900,-176.005,8.391,148.495
C08792=1193.333,375.149,-78.934,-176.003,8.394,148.496
C08793=1193.330,375.397,-78.968,-176.002,8.396,148.496
C08794=1193.325,375.644,-79.003,-176.001,8.400,148.497
C08795=1193.321,375.893,-79.038,-176.000,8.403,148.497
C08796=1193.318,376.140,-79.071,-175.999,8.406,148.498
C08797=1193.314,376.388,-79.106,-175.997,8.410,148.498
C08798=1193.310,376.635,-79.140,-175.996,8.413,148.499
C08799=1193.305,376.882,-79.175,-175.995,8.416,148.499
C08800=1193.301,377.130,-79.209,-175.994,8.418,148.500
C08801=1193.297,377.378,-79.243,-175.992,8.422,148.500
C08802=1193.294,377.626,-79.278,-175.991,8.425,148.501
C08803=1193.289,377.873,-79.313,-175.990,8.428,148.501
C08804=1193.286,378.121,-79.347,-175.989,8.431,148.502
C08805=1193.281,378.368,-79.381,-175.988,8.434,148.502
C08806=1193.277,378.616,-79.416,-175.987,8.438,148.503
C08807=1193.273,378.864,-79.450,-175.986,8.441,148.503
C08808=1193.269,379.111,-79.484,-175.985,8.444,148.504
C08809=1193.265,379.358,-79.520,-175.984,8.447,148.504
C08810=1193.261,379.606,-79.555,-175.983,8.450,148.505
C08811=1193.257,379.854,-79.589,-175.982,8.453,148.505
C08812=1193.253,380.101,-79.623,-175.980,8.457,148.506
C08813=1193.249,380.349,-79.658,-175.980,8.460,148.506
C08814=1193.245,380.596,-79.692,-175.978,8.463,148.507
C08815=1193.241,380.844,-79.727,-175.978,8.466,148.507
C08816=1193.237,381.091,-79.762,-175.977,8.469,148.508
C08817=1193.233,381.339,-79.797,-175.976,8.472,148.508
C08818=1193.229,381.587,-79.831,-175.975,8.475,148.509
C08819=1193.225,381.835,-79.865,-175.974,8.478,148.510
C08820=1193.221,382.081,-79.901,-175.973,8.481,148.510
C08821=1193.217,382.330,-79.935,-175.972,8.484,148.511
C08822=1193.213,382.577,-79.969,-175.971,8.487,148.511
C08823=1193.209,382.825,-80.004,-175.970,8.490,148.512
C08824=1193.205,383.072,-80.039,-175.970,8.493,148.512
C08825=1193.201,383.320,-80.074,-175.968,8.496,148.513
C08826=1193.197,383.567,-80.108,-175.968,8.499,148.513
C08827=1193.193,383.815,-80.143,-175.967,8.502,148.514
C08828=1193.189,384.062,-80.178,-175.966,8.505,148.514
C08829=1193.185,384.310,-80.213,-175.965,8.508,148.515
C08830=1193.180,384.557,-80.247,-175.964,8.511,148.515
C08831=1193.177,384.804,-80.282,-175.963,8.514,148.516
C08832=1193.173,385.052,-80.317,-175.962,8.517,148.517
C08833=1193.169,385.300,-80.352,-175.962,8.520,148.517
C08834=1193.165,385.548,-80.387,-175.961,8.523,148.518
C08835=1193.160,385.795,-80.422,-175.961,8.526,148.518
C08836=1193.156,386.043,-80.456,-175.960,8.529,148.519
C08837=1193.153,386.290,-80.491,-175.959,8.532,148.519
C08838=1193.149,386.538,-80.526,-175.958,8.535,148.520
C08839=1193.144,386.785,-80.560,-175.957,8.537,148.520
C08840=1193.141,387.033,-80.596,-175.957,8.540,148.521
C08841=1193.136,387.280,-80.630,-175.956,8.543,148.522
C08842=1193.132,387.527,-80.666,-175.955,8.546,148.522
C08843=1193.128,387.776,-80.701,-175.955,8.548,148.523
C08844=1193.125,388.023,-80.735,-175.954,8.552,148.523
C08845=1193.121,388.270,-80.770,-175.953,8.555,148.524
C08846=1193.116,388.518,-80.805,-175.952,8.558,148.524
C08847=1193.113,388.765,-80.840,-175.952,8.560,148.525
C08848=1193.108,389.013,-80.875,-175.951,8.563,148.526
C08849=1193.105,389.260,-80.910,-175.951,8.566,148.526
C08850=1193.101,389.508,-80.945,-175.950,8.568,148.527
C08851=1193.096,389.756,-80.979,-175.950,8.572,148.527
C08852=1193.092,390.003,-81.015,-175.949,8.575,148.528
C08853=1193.088,390.250,-81.049,-175.949,8.577,148.528
C08854=1193.085,390.498,-81.084,-175.948,8.580,148.529
C08855=1193.081,390.746,-81.119,-175.948,8.582,148.529
C08856=1193.077,390.993,-81.154,-175.947,8.585,148.530
C08857=1193.073,391.241,-81.189,-175.947,8.588,148.531
C08858=1193.068,391.488,-81.224,-175.946,8.591,148.531
C08859=1193.064,391.736,-81.259,-175.945,8.594,148.532
C08860=1193.060,392.019,-81.300,-175.945,8.596,148.532
C08861=1193.055,392.302,-81.339,-175.944,8.600,148.533
C08862=1193.051,392.585,-81.380,-175.944,8.603,148.534
C08863=1193.047,392.869,-81.421,-175.943,8.606,148.534
C08864=1193.042,393.116,-81.455,-175.943,8.608,148.535
C08865=1193.038,393.364,-81.491,-175.942,8.611,148.536
C08866=1193.034,393.611,-81.525,-175.942,8.614,148.536
C08867=1193.031,393.858,-81.560,-175.941,8.617,148.537
C08868=1193.027,394.106,-81.595,-175.941,8.619,148.537
C08869=1193.023,394.353,-81.630,-175.941,8.622,148.538
C08870=1193.019,394.601,-81.666,-175.940,8.625,148.539
C08871=1193.015,394.849,-81.701,-175.940,8.627,148.539
C08872=1193.011,395.096,-81.736,-175.939,8.630,148.540
C08873=1193.007,395.344,-81.771,-175.939,8.632,148.540
C08874=1193.002,395.591,-81.806,-175.938,8.635,148.541
C08875=1192.999,395.838,-81.841,-175.938,8.638,148.541
C08876=1192.995,396.086,-81.876,-175.938,8.640,148.542
C08877=1192.991,396.333,-81.911,-175.937,8.643,148.543
C08878=1192.987,396.581,-81.946,-175.937,8.646,148.543
C08879=1192.983,396.829,-81.982,-175.937,8.648,148.544
C08880=1192.979,397.075,-82.017,-175.937,8.650,148.544
C08881=1192.975,397.324,-82.052,-175.936,8.653,148.545
C08882=1192.971,397.571,-82.087,-175.936,8.656,148.545
C08883=1192.966,397.818,-82.123,-175.935,8.658,148.546
C08884=1192.962,398.066,-82.158,-175.935,8.661,148.546
C08885=1192.958,398.314,-82.193,-175.935,8.663,148.547
C08886=1192.954,398.561,-82.229,-175.935,8.666,148.548
C08887=1192.950,398.809,-82.263,-175.934,8.668,148.548
C08888=1192.947,399.056,-82.299,-175.934,8.670,148.549
C08889=1192.942,399.303,-82.334,-175.933,8.673,148.549
C08890=1192.939,399.550,-82.370,-175.933,8.676,148.550
C08891=1192.935,399.799,-82.405,-175.933,8.678,148.550
C08892=1192.930,400.045,-82.440,-175.933,8.680,148.551
C08893=1192.927,400.293,-82.475,-175.933,8.683,148.552
C08894=1192.923,400.541,-82.510,-175.932,8.686,148.552
C08895=1192.918,400.788,-82.545,-175.932,8.688,148.553
C08896=1192.915,401.035,-82.581,-175.931,8.690,148.553
C08897=1192.911,401.283,-82.616,-175.931,8.693,148.554
C08898=1192.907,401.530,-82.651,-175.931,8.695,148.554
C08899=1192.903,401.778,-82.686,-175.931,8.697,148.555
C08900=1192.898,402.026,-82.723,-175.931,8.699,148.555
C08901=1192.895,402.273,-82.758,-175.931,8.702,148.556
C08902=1192.891,402.520,-82.793,-175.930,8.704,148.557
C08903=1192.887,402.768,-82.828,-175.930,8.707,148.557
C08904=1192.883,403.015,-82.864,-175.929,8.710,148.558
C08905=1192.879,403.262,-82.899,-175.929,8.712,148.558
C08906=1192.875,403.510,-82.934,-175.929,8.714,148.559
C08907=1192.871,403.758,-82.969,-175.929,8.716,148.559
C08908=1192.867,404.005,-83.005,-175.928,8.719,148.560
C08909=1192.863,404.252,-83.040,-175.929,8.721,148.561
C08910=1192.859,404.500,-83.076,-175.928,8.724,148.561
C08911=1192.855,404.748,-83.112,-175.928,8.726,148.562
C08912=1192.850,404.995,-83.146,-175.928,8.728,148.562
C08913=1192.847,405.242,-83.182,-175.928,8.730,148.563
C08914=1192.843,405.490,-83.217,-175.927,8.733,148.563
C08915=1192.839,405.737,-83.253,-175.927,8.735,148.564
C08916=1192.835,405.984,-83.288,-175.927,8.737,148.564
C08917=1192.832,406.232,-83.324,-175.927,8.739,148.565
C08918=1192.827,406.480,-83.360,-175.926,8.742,148.565
C08919=1192.823,406.727,-83.394,-175.927,8.744,148.566
C08920=1192.819,406.974,-83.430,-175.926,8.747,148.567
C08921=1192.815,407.222,-83.465,-175.926,8.749,148.567
C08922=1192.812,407.469,-83.501,-175.926,8.750,148.568
C08923=1192.807,407.716,-83.536,-175.926,8.752,148.568
C08924=1192.803,407.964,-83.572,-175.926,8.755,148.569
C08925=1192.799,408.212,-83.608,-175.926,8.757,148.569
C08926=1192.795,408.460,-83.642,-175.926,8.759,148.570
C08927=1192.791,408.706,-83.678,-175.925,8.762,148.570
C08928=1192.787,408.954,-83.713,-175.925,8.764,148.571
C08929=1192.784,409.201,-83.749,-175.925,8.766,148.571
C08930=1192.779,409.449,-83.785,-175.925,8.768,148.572
C08931=1192.775,409.696,-83.820,-175.924,8.771,148.572
C08932=1192.771,409.944,-83.856,-175.925,8.772,148.573
C08933=1192.768,410.191,-83.891,-175.924,8.774,148.573
C08934=1192.764,410.439,-83.927,-175.924,8.777,148.574
C08935=1192.760,410.685,-83.962,-175.924,8.779,148.574
C08936=1192.755,410.933,-83.998,-175.924,8.781,148.575
C08937=1192.752,411.181,-84.034,-175.924,8.784,148.576
C08938=1192.748,411.429,-84.068,-175.924,8.785,148.576
C08939=1192.744,411.676,-84.104,-175.924,8.787,148.577
C08940=1192.740,411.923,-84.139,-175.924,8.790,148.577
C08941=1192.735,412.171,-84.175,-175.923,8.792,148.578
C08942=1192.732,412.418,-84.211,-175.923,8.794,148.578
C08943=1192.728,412.665,-84.246,-175.923,8.796,148.579
C08944=1192.724,412.913,-84.282,-175.923,8.798,148.579
C08945=1192.720,413.160,-84.317,-175.923,8.800,148.580
C08946=1192.716,413.408,-84.353,-175.923,8.802,148.580
C08947=1192.712,413.656,-84.389,-175.922,8.805,148.581
C08948=1192.708,413.902,-84.424,-175.922,8.806,148.581
C08949=1192.704,414.150,-84.460,-175.922,8.808,148.581
C08950=1192.700,414.398,-84.496,-175.922,8.810,148.582
C08951=1192.696,414.645,-84.531,-175.922,8.813,148.583
C08952=1192.692,414.892,-84.566,-175.922,8.814,148.583
C08953=1192.688,415.139,-84.602,-175.922,8.816,148.584
C08954=1192.685,415.387,-84.638,-175.921,8.819,148.584
C08955=1192.680,415.635,-84.674,-175.921,8.821,148.585
C08956=1192.674,416.005,-84.727,-175.921,8.823,148.585
C08957=1192.671,416.375,-84.780,-175.921,8.827,148.586
C08958=1192.669,416.745,-84.833,-175.921,8.829,148.587
C08959=1192.673,417.114,-84.885,-175.920,8.832,148.587
C08960=1192.251,417.114,-84.925,-175.923,8.843,148.591
C08961=1192.248,416.742,-84.872,-175.924,8.840,148.590
C08962=1192.249,416.370,-84.819,-175.924,8.837,148.590
C08963=1192.252,415.997,-84.765,-175.924,8.834,148.589
C08964=1192.259,415.624,-84.712,-175.924,8.831,148.588
C08965=1192.263,415.376,-84.676,-175.925,8.829,148.588
C08966=1192.267,415.128,-84.641,-175.925,8.827,148.587
C08967=1192.271,414.881,-84.605,-175.925,8.825,148.587
C08968=1192.274,414.633,-84.570,-175.925,8.823,148.586
C08969=1192.279,414.386,-84.534,-175.925,8.821,148.586
C08970=1192.283,414.139,-84.498,-175.925,8.819,148.585
C08971=1192.287,413.891,-84.463,-175.925,8.816,148.585
C08972=1192.290,413.644,-84.427,-175.925,8.815,148.584
C08973=1192.295,413.397,-84.392,-175.925,8.813,148.584
C08974=1192.299,413.149,-84.356,-175.926,8.810,148.583
C08975=1192.303,412.902,-84.320,-175.926,8.808,148.583
C08976=1192.306,412.654,-84.285,-175.926,8.807,148.582
C08977=1192.310,412.407,-84.249,-175.926,8.805,148.582
C08978=1192.315,412.160,-84.213,-175.926,8.802,148.581
C08979=1192.319,411.912,-84.178,-175.926,8.800,148.581
C08980=1192.322,411.665,-84.142,-175.927,8.798,148.580
C08981=1192.326,411.417,-84.107,-175.926,8.796,148.580
C08982=1192.330,411.170,-84.072,-175.926,8.794,148.579
C08983=1192.335,410.923,-84.035,-175.927,8.792,148.579
C08984=1192.338,410.675,-84.000,-175.927,8.789,148.578
C08985=1192.342,410.428,-83.964,-175.927,8.787,148.577
C08986=1192.346,410.181,-83.929,-175.927,8.785,148.577
C08987=1192.350,409.933,-83.894,-175.927,8.784,148.576
C08988=1192.354,409.685,-83.858,-175.927,8.781,148.576
C08989=1192.358,409.437,-83.823,-175.928,8.779,148.575
C08990=1192.362,409.191,-83.787,-175.928,8.777,148.575
C08991=1192.366,408.943,-83.752,-175.928,8.774,148.574
C08992=1192.370,408.696,-83.716,-175.928,8.772,148.574
C08993=1192.373,408.448,-83.681,-175.929,8.770,148.573
C08994=1192.378,408.201,-83.645,-175.929,8.768,148.573
C08995=1192.382,407.953,-83.610,-175.929,8.766,148.572
C08996=1192.386,407.706,-83.574,-175.929,8.764,148.572
C08997=1192.389,407.458,-83.538,-175.929,8.761,148.571
C08998=1192.394,407.212,-83.503,-175.929,8.759,148.571
C08999=1192.398,406.963,-83.468,-175.929,8.757,148.570
C09000=1192.402,406.716,-83.432,-175.929,8.755,148.569
C09001=1192.406,406.468,-83.397,-175.930,8.752,148.569
C09002=1192.410,406.221,-83.362,-175.930,8.750,148.568
C09003=1192.414,405.974,-83.326,-175.930,8.748,148.568
C09004=1192.417,405.726,-83.290,-175.930,8.746,148.567
C09005=1192.421,405.479,-83.255,-175.931,8.743,148.567
C09006=1192.426,405.231,-83.220,-175.931,8.741,148.566
C09007=1192.430,404.984,-83.184,-175.931,8.738,148.566
C09008=1192.434,404.736,-83.149,-175.931,8.736,148.565
C09009=1192.438,404.489,-83.114,-175.931,8.734,148.565
C09010=1192.442,404.242,-83.078,-175.931,8.732,148.564
C09011=1192.445,403.994,-83.042,-175.932,8.729,148.564
C09012=1192.449,403.746,-83.008,-175.932,8.727,148.563
C09013=1192.453,403.499,-82.972,-175.932,8.725,148.562
C09014=1192.457,403.252,-82.937,-175.932,8.723,148.562
C09015=1192.461,403.004,-82.901,-175.932,8.720,148.561
C09016=1192.466,402.757,-82.866,-175.932,8.718,148.561
C09017=1192.470,402.509,-82.831,-175.933,8.715,148.560
C09018=1192.473,402.262,-82.795,-175.933,8.713,148.560
C09019=1192.477,402.014,-82.760,-175.933,8.711,148.559
C09020=1192.481,401.767,-82.724,-175.933,8.709,148.559
C09021=1192.485,401.519,-82.690,-175.934,8.706,148.558
C09022=1192.489,401.272,-82.654,-175.934,8.703,148.557
C09023=1192.493,401.025,-82.619,-175.934,8.701,148.557
C09024=1192.497,400.777,-82.583,-175.934,8.698,148.556
C09025=1192.501,400.529,-82.549,-175.935,8.696,148.556
C09026=1192.505,400.283,-82.513,-175.935,8.694,148.555
C09027=1192.510,400.035,-82.477,-175.935,8.692,148.555
C09028=1192.513,399.787,-82.442,-175.936,8.689,148.554
C09029=1192.518,399.540,-82.407,-175.936,8.686,148.554
C09030=1192.521,399.292,-82.372,-175.936,8.684,148.553
C09031=1192.525,399.045,-82.336,-175.936,8.681,148.552
C09032=1192.529,398.798,-82.301,-175.936,8.679,148.552
C09033=1192.533,398.550,-82.266,-175.937,8.676,148.551
C09034=1192.537,398.302,-82.231,-175.938,8.674,148.551
C09035=1192.541,398.055,-82.195,-175.938,8.672,148.550
C09036=1192.545,397.807,-82.161,-175.938,8.669,148.550
C09037=1192.549,397.560,-82.125,-175.938,8.666,148.549
C09038=1192.553,397.313,-82.090,-175.939,8.664,148.548
C09039=1192.557,397.065,-82.055,-175.939,8.661,148.548
C09040=1192.561,396.818,-82.019,-175.939,8.659,148.547
C09041=1192.565,396.571,-81.984,-175.940,8.656,148.547
C09042=1192.569,396.323,-81.949,-175.940,8.654,148.546
C09043=1192.573,396.075,-81.914,-175.940,8.651,148.546
C09044=1192.577,395.828,-81.879,-175.941,8.648,148.545
C09045=1192.581,395.580,-81.844,-175.941,8.646,148.544
C09046=1192.585,395.333,-81.808,-175.941,8.644,148.544
C09047=1192.589,395.085,-81.774,-175.942,8.640,148.543
C09048=1192.593,394.838,-81.738,-175.942,8.638,148.543
C09049=1192.596,394.590,-81.703,-175.942,8.636,148.542
C09050=1192.601,394.343,-81.668,-175.943,8.633,148.541
C09051=1192.605,394.095,-81.633,-175.944,8.631,148.541
C09052=1192.609,393.847,-81.598,-175.944,8.627,148.540
C09053=1192.613,393.600,-81.563,-175.944,8.625,148.540
C09054=1192.617,393.353,-81.527,-175.945,8.622,148.539
C09055=1192.621,393.106,-81.493,-175.945,8.620,148.539
C09056=1192.625,392.858,-81.457,-175.945,8.617,148.538
C09057=1192.630,392.574,-81.417,-175.946,8.614,148.537
C09058=1192.634,392.292,-81.377,-175.947,8.611,148.537
C09059=1192.639,392.008,-81.337,-175.947,8.608,148.536
C09060=1192.643,391.724,-81.296,-175.948,8.604,148.535
C09061=1192.648,391.477,-81.262,-175.948,8.602,148.535
C09062=1192.651,391.229,-81.226,-175.949,8.599,148.534
C09063=1192.655,390.981,-81.192,-175.950,8.596,148.534
C09064=1192.659,390.734,-81.156,-175.950,8.594,148.533
C09065=1192.663,390.487,-81.122,-175.951,8.590,148.532
C09066=1192.667,390.240,-81.087,-175.951,8.588,148.532
C09067=1192.671,389.992,-81.052,-175.952,8.585,148.531
C09068=1192.675,389.744,-81.017,-175.952,8.582,148.531
C09069=1192.679,389.497,-80.982,-175.953,8.580,148.530
C09070=1192.683,389.249,-80.947,-175.953,8.577,148.530
C09071=1192.687,389.002,-80.912,-175.954,8.574,148.529
C09072=1192.691,388.754,-80.877,-175.954,8.571,148.528
C09073=1192.696,388.507,-80.842,-175.955,8.568,148.528
C09074=1192.699,388.259,-80.807,-175.956,8.565,148.527
C09075=1192.702,388.012,-80.772,-175.956,8.563,148.527
C09076=1192.707,387.765,-80.737,-175.957,8.560,148.526
C09077=1192.711,387.517,-80.702,-175.958,8.557,148.526
C09078=1192.715,387.269,-80.668,-175.958,8.554,148.525
C09079=1192.719,387.022,-80.632,-175.959,8.551,148.524
C09080=1192.723,386.774,-80.597,-175.960,8.548,148.524
C09081=1192.727,386.527,-80.562,-175.960,8.545,148.523
C09082=1192.731,386.279,-80.527,-175.961,8.542,148.523
C09083=1192.735,386.032,-80.494,-175.962,8.540,148.522
C09084=1192.739,385.784,-80.458,-175.962,8.537,148.522
C09085=1192.743,385.537,-80.424,-175.964,8.534,148.521
C09086=1192.747,385.289,-80.389,-175.964,8.531,148.521
C09087=1192.751,385.042,-80.354,-175.965,8.528,148.520
C09088=1192.755,384.794,-80.319,-175.966,8.524,148.519
C09089=1192.759,384.547,-80.285,-175.967,8.521,148.519
C09090=1192.763,384.299,-80.249,-175.968,8.518,148.518
C09091=1192.767,384.051,-80.214,-175.968,8.516,148.518
C09092=1192.771,383.804,-80.180,-175.969,8.513,148.517
C09093=1192.775,383.556,-80.144,-175.970,8.510,148.517
C09094=1192.779,383.309,-80.111,-175.971,8.507,148.516
C09095=1192.783,383.061,-80.076,-175.971,8.504,148.516
C09096=1192.787,382.814,-80.041,-175.972,8.501,148.515
C09097=1192.791,382.566,-80.006,-175.973,8.498,148.515
C09098=1192.795,382.319,-79.972,-175.974,8.495,148.514
C09099=1192.799,382.071,-79.937,-175.975,8.492,148.513
C09100=1192.803,381.824,-79.902,-175.976,8.489,148.513
C09101=1192.807,381.576,-79.867,-175.977,8.486,148.512
C09102=1192.811,381.329,-79.833,-175.978,8.483,148.512
C09103=1192.815,381.081,-79.798,-175.979,8.479,148.511
C09104=1192.820,380.833,-79.764,-175.980,8.476,148.511
C09105=1192.823,380.586,-79.728,-175.981,8.473,148.510
C09106=1192.827,380.339,-79.694,-175.982,8.470,148.510
C09107=1192.831,380.090,-79.660,-175.983,8.467,148.509
C09108=1192.836,379.843,-79.625,-175.984,8.464,148.509
C09109=1192.840,379.595,-79.590,-175.985,8.461,148.508
C09110=1192.843,379.348,-79.556,-175.986,8.458,148.508
C09111=1192.847,379.100,-79.521,-175.987,8.454,148.507
C09112=1192.852,378.853,-79.486,-175.988,8.451,148.507
C09113=1192.855,378.606,-79.453,-175.989,8.448,148.506
C09114=1192.859,378.358,-79.418,-175.990,8.445,148.506
C09115=1192.864,378.110,-79.383,-175.991,8.442,148.505
C09116=1192.867,377.862,-79.349,-175.993,8.438,148.505
C09117=1192.872,377.615,-79.315,-175.994,8.436,148.504
C09118=1192.876,377.367,-79.280,-175.995,8.432,148.504
C09119=1192.880,377.120,-79.246,-175.996,8.430,148.503
C09120=1192.884,376.872,-79.211,-175.997,8.426,148.503
C09121=1192.888,376.624,-79.177,-175.999,8.423,148.502
C09122=1192.892,376.378,-79.142,-175.999,8.420,148.502
C09123=1192.896,376.130,-79.107,-176.001,8.417,148.501
C09124=1192.900,375.882,-79.073,-176.002,8.413,148.501
C09125=1192.903,375.634,-79.038,-176.003,8.410,148.500
C09126=1192.908,375.387,-79.004,-176.004,8.408,148.500
C09127=1192.911,375.139,-78.970,-176.006,8.404,148.499
C09128=1192.916,374.892,-78.935,-176.007,8.401,148.499
C09129=1192.920,374.644,-78.901,-176.008,8.398,148.498
C09130=1192.924,374.396,-78.867,-176.010,8.394,148.498
C09131=1192.928,374.148,-78.833,-176.011,8.391,148.497
C09132=1192.932,373.901,-78.799,-176.012,8.388,148.497
C09133=1192.936,373.653,-78.764,-176.013,8.385,148.496
C09134=1192.941,373.406,-78.730,-176.015,8.382,148.496
C09135=1192.944,373.158,-78.695,-176.016,8.378,148.495
C09136=1192.949,372.911,-78.661,-176.017,8.375,148.495
C09137=1192.952,372.663,-78.627,-176.018,8.372,148.495
